// TIA Portal V20 program export: 4 tag tables, 69 data types, 13 data blocks, 100 code blocks (in call order from the OBs), 16 instance data blocks

VAR_GLOBAL   // PLC tag table "Default tag table"
END_VAR

VAR_GLOBAL   // PLC tag table "LKinCtrl_Configuration"
END_VAR
VAR_GLOBAL CONSTANT   // user constants
   LKINCTRL_SPTP_EXECUTION_STATUS_OUTPUT : Int := 0;   // 0: Regular time status; 1: Inverted time status; 2: Approximate cartesian distance
   LKINCTRL_LENGTH_OF_OFFSET_NAME : Int := 20;   // Length of offset name
   LKINCTRL_DISABLE_FLAG_RESET : Bool := TRUE;   // FALSE: Reset with execute & after done ; TRUE: No reset
   LKINCTRL_NO_OF_OFFSETS : Int := 3;   // Number of configurable offsets
   LKINCTRL_NO_OF_START_EXECUTE_CMDS : Int := 1;   // Number of cmds to be buffered in first cycle
   LKINCTRL_LENGTH_OF_CMDPOINT_NAME : Int := 30;   // Length of point name
   LKINCTRL_NO_OF_CONVEYOR : Int := 5;   // Number of configurable offsets
   LKINCTRL_NO_OF_SEQ_EXECUTE_CMDS : Int := 1;   // Number of cmds to be buffered after first cycle
   LKINCTRL_NO_OF_CMD_VALUEFLAGS : Int := 4;   // Number of LREAL flags per command
   LKINCTRL_NO_OF_ZONES : Int := 10;   // Number of zone definitions
   LKINCTRL_NO_OF_PATHDATA_ELEMENTS : Int := 200;   // Length of LKinCtrl_typePathData
   LKINCTRL_NO_OF_CMD_SETFLAGS : Int := 3;   // Number of Boolean flags per command
   LKINCTRL_LENGTH_OF_PATHDATA_NAME : Int := 20;   // Length of PathData name
   LKINCTRL_NO_OF_POINTS_AT_POINT_TABLE : Int := 30;   // Number of points at point table. Valid values are 1..x
   LKINCTRL_LENGTH_OF_TO_NAME : UInt := 30;   // Maximum number of characters for technology object name.
   LKINCTRL_NO_OF_LAST_VALUEFLAG : Int := 30;   // Number of value flags at MovePath FB
   LKINCTRL_NO_OF_LAST_SETFLAG : Int := 30;   // Number of flags at MovePath FB
   LKINCTRL_NO_OF_PATHS : Int := 5;   // Number of paths. Valid values are 1..x
END_VAR

VAR_GLOBAL   // PLC tag table "LKinCtrl_Constants"
END_VAR
VAR_GLOBAL CONSTANT   // user constants
   LKINCTRL_MC_MOVELINEARREL : Int := 2;   // cmdType for linear relative command
   LKINCTRL_FM_SET_BEFORE_AND_NO_RESET : USInt := 1;   // set flag before cmd and no reset
   LKINCTRL_MC_ACTIVATE_KIN_ZONE : Int := 34;   // cmdType for activating a workspace zone
   LKINCTRL_MC_MOVELINEARABS : Int := 1;   // cmdType for linear absolute command
   LKINCTRL_FM_SET_AFTER_AND_NO_RESET_AND_WAIT_FOR_ACKNOWLEDGE : USInt := 15;   // set flag after cmd and wait for external reset
   LKINCTRL_NO_OF_PATHDATA_PREBUFFER_ELEMENTS : Int := 5;   // number of PreBuffer elements
   LKINCTRL_FM_RESET_BEFORE : USInt := 20;   // reset flag at start of command
   LKINCTRL_FM_NO_SET_AND_WAIT_FOR_FALSE_ONCE : USInt := 25;   // do not set or reset flag but wait for flag to be false once during command
   LKINCTRL_TABLE_MASK_ARRAY_ENTRIES : DInt := 10;   // maximum size of searchable table
   LKINCTRL_CS_USER_FRAME_4 : Int := 14;   // select fourth user frame
   LKINCTRL_MC_MOVEDIRECTREL : Int := 6;   // cmdType for move direct relative command
   LKINCTRL_FM_DEACTIVATED : USInt := 0;   // flag deactiavted
   LKINCTRL_FM_SET_BEFORE_AND_RESET_AFTER_ONE_CYCLE : USInt := 3;   // set flag before cmd and reset after one cycle
   LKINCTRL_MC_SET_USER_FRAME : Int := 21;   // cmdType for set user frame
   LKINCTRL_CS_NO_OF_FIRST_USER_FRAME : Int := 11;   // index of first user frame
   LKINCTRL_CONFIG_END_OFFSET_COMP : Int := 40;   // cmdType for ending offset compensation
   LKINCTRL_CMD_WAIT_TIME : Int := 100;   // cmdType for wait time command
   LKINCTRL_COMP_RIGHT : Int := 2;   // tool radius compensation to the right
   LKINCTRL_MC_DEFINE_KIN_ZONE : Int := 33;   // cmdType for definining workspace zone
   LKINCTRL_MC_DESYNC_CONVEYOR : Int := 50;   // cmdType for conveyor desync
   LKINCTRL_MC_ACTIVATE_TOOL : Int := 23;   // cmdType for activating a tool
   LKINCTRL_MC_MOVECIRCULARABS : Int := 3;   // cmdType for circular absolute command
   LKINCTRL_CS_USER_FRAME_3 : Int := 13;   // select third user frame
   LKINCTRL_NO_OF_SETFLAGS_BUFFER_ELEMENTS : Int := 15;   // set as double of LKINCTRL_NO_OF_PATHDATA_PREBUFFER_ELEMENTS
   LKINCTRL_TABLE_TYPE_NONSELECTABLE : USInt := 2;   // constant for type non selectable table
   LKINCTRL_CS_USER_FRAME_2 : Int := 12;   // select second user frame
   LKINCTRL_CIRCMODE_GCODE : Int := 3;   // circMode used in GCode
   LKINCTRL_FM_SET_BEFORE_AND_NO_RESET_AND_WAIT_FOR_ACKNOWLEDGE : USInt := 5;   // set flag before cmd and wait for external reset
   LKINCTRL_CS_NO_OF_LAST_USER_FRAME : Int := 15;   // index of last user frame
   LKINCTRL_MC_ACTIVATE_WS_ZONE : Int := 31;   // cmdType for activating a workspace zone
   LKINCTRL_CS_USER_FRAME_1 : Int := 11;   // select first user frame
   LKINCTRL_MC_DEACTIVATE_WS_ZONE : Int := 32;   // cmdType for deactivating workspace zone
   LKINCTRL_FM_DISTANCE_TOLERANCE : LReal := 0.01;   // tolerance for flagmode 10
   LKINCTRL_CONFIG_START_OFFSET_COMP_LEFT : Int := 41;   // cmdType for starting offset compensation left
   LKINCTRL_FM_SET_BEFORE_AND_RESET_AFTER : USInt := 2;   // set flag before cmd and reset after
   LKINCTRL_MC_MOVECIRCULARREL : Int := 4;   // cmdType for circular relative command
   LKINCTRL_OUTER_CORNER : Int := 1;   // Outer corner (linear / linear intersection)
   LKINCTRL_INNER_CORNER : Int := 2;   // Inner corner (linear / linear intersection)
   LKINCTRL_FM_NO_SET_AND_WAIT_FOR_TRUE_ONCE : USInt := 26;   // do not set or reset flag but wait for flag to be true once during command
   LKINCTRL_MC_SHIFT_CS_REL : Int := 60;   // cmdType for relative shift of CS
   LKINCTRL_FM_SET_AT_REMAINING_DISTANCE : USInt := 10;   // set flag at remaining distance
   LKINCTRL_MC_DEACTIVATE_KIN_ZONE : Int := 35;   // cmdType for deactivating workspace zone
   LKINCTRL_COMP_LEFT : Int := 1;   // tool radius compensation to the left
   LKINCTRL_FM_SET_AFTER_AND_RESET_AFTER_ONE_CYCLE : USInt := 13;   // set flag after cmd and reset after one cycle
   LKINCTRL_CONFIG_START_OFFSET_COMP_RIGHT : Int := 42;   // cmdType for starting offset compensation right
   LKINCTRL_CS_USER_FRAME_5 : Int := 15;   // select fifth user frame
   LKINCTRL_TABLE_TYPE_SELECTABLE : USInt := 1;   // constant for type regular table
   LKINCTRL_MC_TRACKCONVEYORBELT : Int := 10;   // cmdType for track conveyor belt command
   LKINCTRL_NO_OF_VALID_BITS : Int := 6;   // number of valid bits in PathDataElement_advanced
   LKINCTRL_MC_SET_OCS_FRAME : Int := 20;   // cmdType for set frame command
   LKINCTRL_FM_SET_AFTER_AND_NO_RESET : USInt := 11;   // set flag after cmd and no reset
   LKINCTRL_MC_MOVEDIRECTABS : Int := 5;   // cmdType for move direct absolute command
   LKINCTRL_CMD_FLAG_ONLY : Int := 0;   // cmdType for flagOnly command (no motion)
   LKINCTRL_MC_DEFINE_WS_ZONE : Int := 30;   // cmdType for definining workspace zone
   LKINCTRL_MC_RESET_SHIFT : Int := 61;   // cmdType for resetting relative shift of CS
   LKINCTRL_FM_RESET_AFTER : USInt := 21;   // reset flag at end of command
   LKINCTRL_PI : LReal := 3.1415926535897932846264;   // constant value for pi
   LKINCTRL_FM_RESET_AT_REMAINING_DISTANCE : USInt := 22;   // reset flag if remaining distance of current command is reached
   LKINCTRL_MC_MOVELINEARPICKANDPLACE : Int := 11;   // cmdType for linear pick and place command sequence
   LKINCTRL_MC_SET_TOOL_FRAME : Int := 22;   // cmdType for defining tool frame
   LKINCTRL_DEFAULT_TO_NAME : WString := '- - -';   // Default name for technology objects
   LKINCTRL_KINEMATICS_TCS : DInt := 3;
   LKINCTRL_KINEMATICS_KINEMATICSZONES : DInt := 10;
   LKINCTRL_KINEMATICS_ZONE_STATE_VIOLATED : UInt := 3;   // Zone is valid, active and violated
   LKINCTRL_KINEMATICS_ZONE_STATE_INVALID : UInt := 0;   // Zone is invalid, inactive and not violated
   LKINCTRL_KINEMATICS_ZONE_STATE_VALID : UInt := 1;   // Zone is valid but not inactive and not violated
   LKINCTRL_KINEMATICS_WORKSPACEZONES : DInt := 10;
   LKINCTRL_KINEMATICS_OCS : DInt := 3;
   LKINCTRL_KINEMATICS_ZONE_STATE_ACTIVE : UInt := 2;   // Zone is valid and active but not violated
   LKINCTRL_KINEMATICS_CONVEYOR_TRACKING : UInt := 3;
   LKINCTRL_KINEMATICS_AXES : DInt := 6;
   LKINCTRL_MEAS_CMD_WITH_ACK : USInt := 2;   // continue after measurement command only with acknowledge
   LKINCTRL_MEAS_CMD_WO_ACK : USInt := 1;   // continue after measurement command without acknowledge
   LKINCTRL_DEFAULT_NAME : WString := '- - -';   // default name of points in datatype
   LKINCTRL_DEFAULT_NAME_STRING : String := '- - -';   // default name of strings in datatype
   LKINCTRL_NO_OF_PATHDATA_ELEMENTS_ADVANCED : Int := 200;   // LEGACY / Length of LKinCtrl_typePathData_advanced
   LKINCTRL_NO_OF_PATHDATA_ELEMENTS_REDUCED : Int := 10;   // LEGACY / Length of LKinCtrl_typePathData_reduced
END_VAR

VAR_GLOBAL   // PLC tag table "MC_Constants"
END_VAR
VAR_GLOBAL CONSTANT   // user constants
   DIRA_POSITIVE : Int := 1;   // Orientation direction 1: Positive direction
   DA_DEACTIVATED : Int := 0;   // Dynamic adaption 0: Deactivated
   CS_MCS : Int := 100;   // Coordinate system 100: Machine coordinate system (axis values)
   SM_ACTIVE_DYNAMICS : Int := 0;   // Stop mode 0: Stop with active dynamics
   LC_DEFAULT : DWord := 16#FFFFFFFF;   // LinkConstellation: Default to keep link constellation of kinematics
   CM_CENTER : Int := 1;   // Circle mode 1: "Arc" + "AuxPoint" defines circle center
   ZONE_DEACTIVATION_MODE_SIGNAL : DInt := 3;   // Zone deactivation mode 3: All signal zones
   BM_BLENDING_HIGH : Int := 5;   // Buffer mode 5: Blending with higher velocity
   BM_BUFFERED : Int := 1;   // Buffer mode 1: Standstill between motions
   PC_LONG_RUN_POSITIVE : Int := 2;   // Path choice 2: Longer positive circle segment
   IM_MAX_DYNAMICS : Int := 1;   // Interrupt mode 1: Interrupt with maximum dynamics
   CS_FCS : DInt := 0;   // Coordinate system 0: Flange coordinate system (FCS); Only valid for kinematics zone commands
   CS_TCS : DInt := 1;   // Coordinate system 1: Tool coordinate system (TCS); Only valid for kinematics zone commands
   DA_WITH_VARIABLE_LIMITS : Int := 1;   // Dynamic adaption 1: With segmentation of path
   DIRA_SHORTEST : Int := 3;   // Orientation direction 3: Shortest direction
   CS_OCS3 : Int := 3;   // Coordinate system 3: Object coordinate system 3 (OCS[3])
   CS_OCS1 : Int := 1;   // Coordinate system 1: Object coordinate system 1 (OCS[1])
   CM_RADIUS : Int := 2;   // Circle mode 2: "Radius" + "EndPoint" parameters define the circle segment
   CM_BORDER : Int := 0;   // Circle mode 0: "EndPoint" + "AuxPoint" parameter defines a point on circular path
   SM_MAX_DYNAMICS : Int := 1;   // Stop mode 1: Stop with maximum dynamics
   CP_XZ : Int := 0;   // Circle plane 0: Circle in X-Z plane
   CP_YZ : Int := 1;   // Circle plane 1: Circle in Y-Z plane
   IM_ACTIVE_DYNAMICS : Int := 0;   // Interrupt mode 0: Interrupt with active dynamics
   ZONE_DEACTIVATION_MODE_SPECIFIC : DInt := 0;   // Zone deactivation mode 0: Specific zone index
   BM_BLENDING_LOW : Int := 2;   // Buffer mode 2: Blending with lower velocity
   ZONE_DEACTIVATION_MODE_BLOCKED : DInt := 2;   // Zone deactivation mode 2: All blocked zones
   PC_NEGATIVE : Int := 1;   // Path choice 1: Shorter negative circle segment
   CP_XY : Int := 2;   // Circle plane 2: Circle in X-Y plane
   PM_ABS_ABS : DInt := 1;   // PositionMode 1: Interpretation of cartesian orientation as absolute (only effective for absolute MoveDirect commands)
   DA_WITH_CONSTANT_LIMITS : Int := 2;   // Dynamic adaption 2: No segmentation of path
   CS_OCS2 : Int := 2;   // Coordinate system 2: Object coordinate system 2 (OCS[2])
   CS_JCS : Int := 101;   // Coordinate system 101: Joint coordinate system (joint values)
   ZONE_DEACTIVATION_MODE_WORKSPACE : DInt := 4;   // Zone deactivation mode 4: Currently active workspace zone
   PM_ABS_REL : DInt := 2;   // PositionMode 2: Interpretation of cartesian orientation as relative (only effective for absolute MoveDirect commands)
   DIRA_NEGATIVE : Int := 2;   // Orientation direction 2: Negative direction
   CS_WCS : Int := 0;   // Coordinate system 0: World coordinate system (WCS)
   ZONE_DEACTIVATION_MODE_ALL : DInt := 1;   // Zone deactivation mode 1: All zones
   PC_POSITIVE : Int := 0;   // Path choice 0: Shorter positive circle segment
   PC_LONG_RUN_NEGATIVE : Int := 3;   // Path choice 3: Longer negative circle segment
   DA_DEFAULT : Int := -1;   // Dynamic adaption -1: Use default
END_VAR

TYPE "UDT_PathCmd"
TITLE = Buffered-path command element (V4.0 palletizing)
// One command in the buffered-path command list (GDB_PalletizingPath.aCmd). Authored by FB_AutoCtrl_Palletizing REGION 1, executed by REGION 4.
   STRUCT
      i16_CmdType : Int;   // Command type: 0 = END_OF_PATH, 1 = MOVE, 2 = GRIPPER, 3 = WAIT_ARRIVAL
      x : LReal;   // MOVE: target Cartesian X [mm]
      y : LReal;   // MOVE: target Cartesian Y [mm]
      z : LReal;   // MOVE: target Cartesian Z [mm]
      "a" : LReal;   // MOVE: target wrist orientation A [deg]
      lr_Velocity : LReal;   // MOVE: path velocity [mm/s]
      i16_BufferMode : Int;   // MOVE: MC_MoveLinearAbsolute BufferMode for this command -- 1 = stop at this point (BM_BUFFERED), 5 = blend through it (BM_BLENDING_HIGH). Never 0 (MC_Aborting is invalid for a kinematic path -> 16#80B2).
      lr_DwellMs : LReal;   // GRIPPER: grip/release settle hold time [ms]
      bo_GripperGrip : Bool;   // GRIPPER: level value written to GDB_Control.bo_gripperGrip
      bo_GripperRelease : Bool;   // GRIPPER: if TRUE, pulse GDB_Control.bo_gripperRelease for the dwell then drop it
      bo_IsBoxEnd : Bool;   // MOVE: TRUE on the PLACE_RETRACT move that completes a box -- increments statBoxesPlaced and re-arms the spawn request
      i16_HmiStep : Int;   // Value published to GDB_PalletizingCmd.i16_PalletStep when this command becomes active -- preserves the HMI 1..48 step display
   END_STRUCT;
END_TYPE

TYPE "UDT_Recipe"
TITLE = Box-product recipe (Module D)
// SCARA Phase 2 Module D recipe (2026-05-23). One flat box-product recipe: product L/W/H + gap, pallet base L/W + layer count, palletizing move dynamics. LPallPatt-shaped (typeProductData / typePalletData / typePnPDynamics, pruned for 1511T -- no block-packing, no mirroring, no interlayers, no multigripper). Consumed by FB_PatternAutoGen, which auto-fits a one-block grid and writes the result into GDB_PalletizingCmd's Module-C config members. PSC binds to GDB_ActiveRecipe.recipe.* member-for-member; the recipe library lives HMI-side on the panel.
   STRUCT
      sName : String[32];   // Recipe name (HMI display / identity).
      bo_Valid : Bool := FALSE;   // PSC handshake: PSC sets FALSE before transferring a parameter set and TRUE only after all members are written. FB_PatternAutoGen consumes the recipe only when this is TRUE -- closes the mid-write race that bites v9's recipe adapter.
      product : Struct
         lr_Length : LReal;   // Box length [mm]. Drives pitchX (= lr_Length + lr_Gap) via FB_PatternAutoGen.
         lr_Width : LReal;   // Box width [mm]. Drives pitchY (= lr_Width + lr_Gap).
         lr_Height : LReal;   // Box height [mm] -- copied straight to GDB_PalletizingCmd.lr_BoxHeight, the layer Z spacing for the Module-C builder.
         lr_Gap : LReal;   // Clearance between boxes [mm]; added to box dims to derive pitch. Set 0 for boxes edge-to-edge.
      END_STRUCT;
      pallet : Struct
         lr_BaseLength : LReal;   // Pallet base length [mm]. FB_PatternAutoGen auto-fits how many boxes fit along X: cols = (BaseLength + Gap) DIV (Length + Gap), floored.
         lr_BaseWidth : LReal;   // Pallet base width [mm]. FB_PatternAutoGen auto-fits how many boxes fit along Y: rows = (BaseWidth + Gap) DIV (Width + Gap), floored.
         i16_LayerCount : Int;   // Stacked layers (tower mode -- all layers use the same auto-gen grid). Total boxes = cols x rows x LayerCount, capped at the GDB_PalletizingPath.aCmd[] ceiling (22 for aCmd[1..200]).
      END_STRUCT;
      dynamics : Struct
         lr_Velocity : LReal;   // Palletizing-move path velocity [mm/s]. Written into GDB_PalletizingCmd.lr_MoveVelocity by FB_PatternAutoGen.
         lr_Acceleration : LReal;   // Palletizing-move acceleration [mm/s^2]. Written into GDB_PalletizingCmd.lr_MoveAccel.
         lr_Deceleration : LReal;   // Palletizing-move deceleration [mm/s^2]. Written into GDB_PalletizingCmd.lr_MoveDecel.
         lr_Jerk : LReal;   // Palletizing-move jerk [mm/s^3]. Written into GDB_PalletizingCmd.lr_MoveJerk.
      END_STRUCT;
   END_STRUCT;
END_TYPE

TYPE "UDT_typePoint5"
TITLE = SCARA TCP target point
// SCARA TCP target point (XYZA) for ABCDE 5-point cycle. Wang Shuo / Huashili pattern reference. B/C orientation omitted (SCARA 3D only supports A rotation about Z). / SCARA 末端目标点 (XYZA)，用于 ABCDE 5 点循环。王硕 / 华西丽模式参考。
   STRUCT
      x : LReal := 0.0;   // Cartesian X position [mm] / 笛卡尔 X 坐标 [mm]
      y : LReal := 0.0;   // Cartesian Y position [mm] / 笛卡尔 Y 坐标 [mm]
      z : LReal := 0.0;   // Cartesian Z position [mm] / 笛卡尔 Z 坐标 [mm]
      "a" : LReal := 0.0;   // Wrist orientation rotation A [deg] / 末端旋转角度 A [度]
   END_STRUCT;
END_TYPE

TYPE "UDT_typeMeasureInput"
   STRUCT
      input : Struct
         bo_Active : Bool;
         mode : Int;
      END_STRUCT;
      output : Struct
         done : Bool;
         busy : Bool;
         error : Bool;
         i32_ErrorCode : Word;
         r64_MeasuredValue1 : LReal;
         r64_MeasuredValue2 : LReal;
      END_STRUCT;
   END_STRUCT;
END_TYPE

TYPE "UDT_typePosCtrl"
   STRUCT
      input : Struct
         bo_estop : Bool;
         bo_enable : Bool;
         bo_reset : Bool;
         bo_home : Bool;
         bo_jogforward : Bool;
         bo_jogbackward : Bool;
         bo_movevelocity : Bool;
         bo_posabsolute : Bool;
         bo_posrelative : Bool;
         bo_gearin : Bool;
         bo_camin : Bool;
         bo_camout : Bool;
         bo_halt : Bool;
         bo_stop : Bool;
         configuration : Struct
            home { ExternalWritable := 'False'} : Struct
               i16_mode : Int;
               r64_homeposition : LReal;
               r64_ApproachVelocity : LReal := 10.0;
               r64_ReferencingVelocity : LReal := 5.0;
            END_STRUCT;
            jog : Struct
               r64_velocity : LReal := 5.0;
               r64_acceleration : LReal := 1000.0;
               r64_jerk : LReal := -1.0;
            END_STRUCT;
            movevelocity : Struct
               r64_velocity : LReal := 10.0;
               r64_acceleration : LReal := 1000.0;
               r64_jerk : LReal := -1.0;
               i16_direction : Int;
            END_STRUCT;
            posabsolute : Struct
               r64_velocity : LReal := 10.0;
               r64_position : LReal := 0.0;
               r64_acceleration : LReal := 1000.0;
               r64_jerk : LReal := -1.0;
               i16_direction : Int := 1;
            END_STRUCT;
            posrelative : Struct
               r64_velocity : LReal := 10.0;
               r64_position : LReal := 0.0;
               r64_acceleration : LReal := 1000.0;
               r64_jerk : LReal := -1.0;
            END_STRUCT;
            gearin : Struct
               RatioNumerator : DInt := 1;
               RatioDenominator : DInt := 1;
            END_STRUCT;
            camin : Struct
               i16_syncProfileReference : Int := 2;
               i16_applicationMode : Int := 0;
               r64_masterStartDistance : LReal;
               r64_masterSyncPosition : LReal;
               r64_masterOffset : LReal;
            END_STRUCT;
         END_STRUCT;
      END_STRUCT;
      output : Struct
         bo_communicationOk : Bool;
         bo_enabled : Bool;
         bo_homed : Bool;
         bo_inGear : Bool;
         bo_StarSync : Bool;
         bo_inSync : Bool;
         bo_fault : Bool;
         bo_endprofile : Bool;
         bo_SWLimitMinActived : Bool;
         bo_SWLimitMaxActived : Bool;
         bo_HWLimitMinActived : Bool;
         bo_HWLimitMaxActived : Bool;
         r64_actualVelocity : LReal;
         r64_actualPosition : LReal;
      END_STRUCT;
   END_STRUCT;
END_TYPE

TYPE "UDT_typeSpdCtrl"
   STRUCT
      input : Struct
         bo_enable : Bool := false;
         bo_estop : Bool := false;
         bo_reset : Bool := false;
         r32_speedSet : Real := 0.0;
         r32_torqueLimitSet : Real;
         r32_filterTime : Real := 100.0;
         tCycle : Real := 10.0;
         OBNum : Int := 30;
         HW_IO : HW_IO := 0;
         HW_IO_ADD : HW_IO;
         Reference : Struct
            r32_speed_Rpm : Real;
            r32_Torque_Nm : Real;
            r32_current_A : Real;
            r32_DCVolagte_V : Real;
            r32_power_Kw : Real;
            "r32_temperature_℃" : Real;
         END_STRUCT;
      END_STRUCT;
      output : Struct
         bo_enabled : Bool := false;
         bo_ready : Bool := false;
         bo_driveError : Bool := false;
         r32_actSpeed_Rpm : Real := 0.0;
         r32_actTorque_Nm : Real;
         r32_actCurrent_A : Real;
         r32_actDCVolagte_V : Real;
         r32_actPower_Kw : Real;
         "r32_actTemperature_℃" : Real;
         i16_warningCode : Word;
         i16_faultCode : Word;
      END_STRUCT;
   END_STRUCT;
END_TYPE

TYPE "UDT_typeKinCtrl"
   STRUCT
      input : Struct
         bo_estop : Bool;
         bo_enable : Bool;
         bo_reset : Bool;
         bo_home : Bool;
         jogframe : Struct
            "jogX+" : Bool;
            "jogX-" : Bool;
            "jogY+" : Bool;
            "jogY-" : Bool;
            "jogZ+" : Bool;
            "jogZ-" : Bool;
            "jogA+" : Bool;
            "jogA-" : Bool;
            "jogB+" : Bool;
            "jogB-" : Bool;
            "jogC+" : Bool;
            "jogC-" : Bool;
            bo_jogtoposition : Bool;
         END_STRUCT;
         bo_movepathstart : Bool;
         bo_movepathstop : Bool;
         bo_movepathhalt : Bool;
         configuration : Struct
            home { ExternalWritable := 'False'} : Struct
               i16_mode : Array[1..6] of Int;
               r64_homeposition : Array[1..6] of LReal;
            END_STRUCT;
            jogframe : Struct
               targetposition : Struct
                  x : LReal;
                  y : LReal;
                  z : LReal;
                  "a" : LReal;
                  "b" : LReal;
                  c : LReal;
               END_STRUCT;
               dynamics : "LKinCtrl_typeDynamics";   // Specification of the jog dynamics
            END_STRUCT;
         END_STRUCT;
      END_STRUCT;
      output : Struct
         bo_enabled : Bool;
         bo_homed : Bool;
         bo_fault : Bool;
         bo_done : Bool;
         i16_activeCmdNo : Int;
         actualposition : Struct
            x : LReal;
            y : LReal;
            z : LReal;
            "a" : LReal;
            "b" : LReal;
            c : LReal;
         END_STRUCT;
      END_STRUCT;
      inout : Struct
         PathData { S7_SetPoint := 'True'} : "LKinCtrl_typePathData";
      END_STRUCT;
   END_STRUCT;
   // input.configuration.jogframe.dynamics.sPTP.velocityFactor := -1.0;
   // input.configuration.jogframe.dynamics.sPTP.accelerationFactor := -1.0;
   // input.configuration.jogframe.dynamics.sPTP.decelerationFactor := -1.0;
   // input.configuration.jogframe.dynamics.sPTP.jerkFactor := -1.0;
END_TYPE

TYPE "LKinCtrl_bufferElement"
   STRUCT
      pathDataName : String["LKINCTRL_LENGTH_OF_PATHDATA_NAME"];
      pathDataIdentifier : USInt;
      setNumber : DInt;
      MotionType : Int := -1;
      MotionFBNo : Int;
      coordinateSystem : Int;
      transitionParameter : LReal;
      bufferMode : Int;
      measurementCmd : USInt;
      position : Array[1..6] of LReal;
   END_STRUCT;
END_TYPE

TYPE "LKinCtrl_typeAdvPointers"
   STRUCT
      addPointer : DInt := 0;   // pointer to add new comds to PathData after cmd has been executed by MovePath
      retrievePointer : DInt := 0;   // pointer to show which cmd is the next to be retrieved by MovePath
      addPointerRestarted : Bool;   // addPointer restarted after overflow
      ignoreAddPointer : Bool := TRUE;   // addPointer not taken into account for buffering, unless set by previous data source
      bufferLocked : Bool;   // buffer locked to wait for previous data source - read data locked
      preprocessingStop : Bool;   // parser reached a preprocessing stop
   END_STRUCT;
END_TYPE

TYPE "LKinCtrl_typeAuxFCDiagnostics"
TITLE = typeDiagnosticsFBTemplate
   STRUCT
      status : Word;   // Status of the FB or error identification when error occurred
      subfunctionStatus : Word;   // Status or return value of called FBs, FCs and system blocks
      axisNumber : Int;   // number of the corresponding axis the error occured in or a function effecting it
      errorDetail : UDInt;   // error detail of corresponding technology object the error occured in
      stateNumber : DInt;   // State in the state machine of the FB when the error occurred
   END_STRUCT;
END_TYPE

TYPE "LKinCtrl_typeCartesianPosition"
   STRUCT
      x : LReal;   // X
      y : LReal;   // Y
      z : LReal;   // Z
      "a" : LReal;   // A
      "b" : LReal;   // B
      c : LReal;   // C
   END_STRUCT;
END_TYPE

TYPE "LKinCtrl_typeCircleParameters"
   STRUCT
      circMode : DInt := 0;   // 0: auxPoint defines point on circle line; 1: auxPoint defines circle center; 2: radius and endPoint define circle segment; 3: GCode notation (end & aux point)
      point : DInt := -1;   // reference to point table, used for auxPoint
      auxPoint : Array[1..3] of LReal;   // auxiliary point for circle definition
      pathChoice : DInt := 0;   // circMode(0): not relevant; circMode(1): 0: pos direction; 1: neg direction; circMode(2): 0: short pos segment; 1: short neg segment; 2: long pos segment; 3: long neg segment
      circlePlane : DInt;   // circMode(0): not relevant; circMode(1+2): 0: XZ; 1: YZ; 2: XY
      radius : LReal;   // only in combination with circMode(2): radius
      arc : LReal;   // only in combination with circMode(1): arc
   END_STRUCT;
END_TYPE

TYPE "LKinCtrl_typeCmdLoggerElement"
   STRUCT
      cmdType : Int := -1;   // 1: MoveLinAbs; 2: MoveLinRel; 3: MoveCircAbs; 4: MoveCircRel; 5: MoveDirectAbs; 6: MoveDirectRel; 10: TrackConveyorBelt; 100: WaitTime; 40/41/42: ContourOffset; 0: FlagOnlyCmd; -1: End of List
      pathDataName : String["LKINCTRL_LENGTH_OF_PATHDATA_NAME"];   // name of PathData
      pathDataIdentifier : Int;   // identifier of PathData containing command
      cmdID : DInt;   // to be set to PathDataOperate[list position] by PreBuffer for identification in ExecuteBuffer
      cmdName : String[4];   // command name
      coordinateX : LReal;   // X (linear) / endPoint[1] (circular)
      coordinateY : LReal;   // Y (linear) / endPoint[2] (circular)
      coordinateZ : LReal;   // Z (linear) / endPoint[3] (circular)
      coordinateA : LReal;   // A (linear) / endPoint[4] (circular)
      coordSystem : DInt := 0;   // 0: WCS; 1: OCS[1]; 2: OCS[2]; 3: OCS[3]
      bufferMode : DInt := 1;   // 1: standstill between commands, 2: blending with lower speed; 5: blending with higher speed
      transitionParameter : LReal;   // blending distance - >0.0: configured value used; <0.0: maximum possible blending distance used
      dynVelocity : LReal;   // >0.0: configured value used; <0.0: default TO setting used
      dynAcceleration : LReal;   // >0.0: configured value used; <0.0: default TO setting used
      dynDeceleration : LReal;   // >0.0: configured value used; <0.0: default TO setting used
      dynJerk : LReal;   // >0.0: configured value used; <0.0: default TO setting used
      dynamicAdpation : DInt;   // <0.0: default TO setting used; 0: no dynamic adaption; 1: with variable limits; 2: with constant limits
      linkConstellation : DWord;   // linkConstellation (effective for MoveDirect commands only)
      positionMode : DInt;   // 1: absolute cartesian position and absolute orientation; 2: absolute cartesian position and relative orientation (effective for MoveDirect commands only)
      circMode : DInt;   // 0: auxPoint defines point on circle line; 1: auxPoint defines circle center; 2: radius and endPoint define circle segment
      auxPoint_1 : LReal;   // auxiliary point for circle definition
      auxPoint_2 : LReal;   // auxiliary point for circle definition
      auxPoint_3 : LReal;   // auxiliary point for circle definition
      pathChoice : DInt;   // circMode(0): not relevant; circMode(1): 0: pos direction; 1: neg direction; circMode(2): 0: short pos segment; 1: short neg segment; 2: long pos segment; 3: long neg segment
      circlePlane : DInt;   // circMode(0): not relevant; circMode(1+2): 0: XZ; 1: YZ; 2: XY
      radius : LReal;   // only in combination with circMode(2): radius
      arc : LReal;   // only in combination with circMode(1): arc
   END_STRUCT;
END_TYPE

TYPE "LKinCtrl_typeConfiguration"
   STRUCT
      offsetParameter : Array[1.."LKINCTRL_NO_OF_OFFSETS"] of "LKinCtrl_typeContourOffsetParameter";   // offset parameter settings
      conveyorParameter : Array[1.."LKINCTRL_NO_OF_CONVEYOR"] of "LKinCtrl_typeConveyorConfiguration";   // conveyor parameter settings
      userFrames : Array["LKINCTRL_CS_NO_OF_FIRST_USER_FRAME".."LKINCTRL_CS_NO_OF_LAST_USER_FRAME"] of "LKinCtrl_typeFrame";   // user frames configuration
      workspaceZones : Array[1.."LKINCTRL_NO_OF_ZONES"] of "LKinCtrl_typeWorkspaceZoneDefinition";   // workspace zone configurations
      kinematicsZones : Array[1.."LKINCTRL_NO_OF_ZONES"] of "LKinCtrl_typeKinematicsZoneDefinition";   // kinematics zone configuration
      stopMode : DInt;   // MC_GroupStop dynamics; 0: stop with dynamics of active motion job; 1: stop with maximum kinematics dynamics (dynamics adaption still effective); 10: stop with dynamics of active motion job and desync conveyor; 11: stop with maximum kinematics dynamics and desync conveyor
      interruptMode : DInt;   // MC_GroupInterrupt dynamics; 0: interrupt with dynamics of active motion job; 1: interrupt with maximum kinematics dynamics (dynamics adaption still effective)
   END_STRUCT;
END_TYPE

TYPE "LKinCtrl_typeConfigurationAxis"
   STRUCT
      "name" { ExternalAccessible := 'False'; ExternalVisible := 'False'; ExternalWritable := 'False'; S7_SetPoint := 'True'} : WString["LKINCTRL_LENGTH_OF_TO_NAME"];   // Axis name shown on HMI
      used { ExternalAccessible := 'False'; ExternalVisible := 'False'; ExternalWritable := 'False'; S7_SetPoint := 'True'} : Bool := FALSE;   // TRUE: Axis is used (only relevant for additional axes, kinematic axes are always used)
      withBrake { ExternalAccessible := 'False'; ExternalVisible := 'False'; ExternalWritable := 'False'; S7_SetPoint := 'True'} : Bool := FALSE;   // TRUE: Axis has a motor holding brake
      homePosition { ExternalAccessible := 'False'; ExternalVisible := 'False'; ExternalWritable := 'False'; S7_SetPoint := 'True'} : LReal := 0.0;   // Defines the default homing position
      coupling { ExternalAccessible := 'False'; ExternalVisible := 'False'; ExternalWritable := 'False'; S7_SetPoint := 'True'} : Bool := FALSE;   // TRUE: Coupling present
      jog { ExternalAccessible := 'False'; ExternalVisible := 'False'; ExternalWritable := 'False'; S7_SetPoint := 'True'} : "LKinCtrl_typeJogConfiguration";
   END_STRUCT;
   // jog.accelerationTime := 0.2;
   // jog.maxVelocityManual := 10.0;
   // jog.maxVelocityTestRun := 10.0;
   // jog.presetIncrementCoarse := 5.0;
   // jog.presetIncrementFine := 1.0;
   // jog.presetIncrementPrecise := 0.5;
END_TYPE

TYPE "LKinCtrl_typeConfigurationKinematics"
   STRUCT
      "name" { ExternalAccessible := 'False'; ExternalVisible := 'False'; ExternalWritable := 'False'; S7_SetPoint := 'True'} : WString["LKINCTRL_LENGTH_OF_TO_NAME"];
      jogPath { ExternalAccessible := 'False'; ExternalVisible := 'False'; ExternalWritable := 'False'; S7_SetPoint := 'True'} : "LKinCtrl_typeJogConfiguration";
      jogOrientation { ExternalAccessible := 'False'; ExternalVisible := 'False'; ExternalWritable := 'False'; S7_SetPoint := 'True'} : "LKinCtrl_typeJogConfiguration";
   END_STRUCT;
   // jogPath.accelerationTime := 0.2;
   // jogPath.maxVelocityManual := 250.0;
   // jogPath.maxVelocityTestRun := 250.0;
   // jogPath.presetIncrementCoarse := 10.0;
   // jogPath.presetIncrementFine := 1.0;
   // jogPath.presetIncrementPrecise := 0.1;
   // jogOrientation.accelerationTime := 0.2;
   // jogOrientation.maxVelocityManual := 10.0;
   // jogOrientation.maxVelocityTestRun := 10.0;
   // jogOrientation.presetIncrementCoarse := 5.0;
   // jogOrientation.presetIncrementFine := 1.0;
   // jogOrientation.presetIncrementPrecise := 0.1;
END_TYPE

TYPE "LKinCtrl_typeContourOffsetParameter"
   STRUCT
      "name" : String["LKINCTRL_LENGTH_OF_OFFSET_NAME"];   // offset name
      radius : LReal;   // offset radius
      length : LReal;   // offset length
   END_STRUCT;
END_TYPE

TYPE "LKinCtrl_typeConveyorConfiguration"
   STRUCT
      conveyorBeltAxis : DB_ANY;   // Conveyor belt axis DB
      conveyorBeltOrigin : TO_Struct_Kinematics_Frame;   // Frame to origin of conveyor belt
      initialObjectPosition : TO_Struct_Kinematics_Frame;   // Initial object position on conveyor (only x allowed)
   END_STRUCT;
END_TYPE

TYPE "LKinCtrl_typeConveyorParameter"
   STRUCT
      conveyorParaNo : DInt := 0;   // selection of conveyor parameter set from configuration structure
   END_STRUCT;
END_TYPE

TYPE "LKinCtrl_typeDiagnosticsPathSelect"
TITLE = typeDiagnosticsFBTemplate
   STRUCT
      status : Word;   // Status of the FC or error identification when error occurred
      entryID : Int;   // identifier for false entry
   END_STRUCT;
END_TYPE

TYPE "LKinCtrl_typeDynamics"
   STRUCT
      path : "LKinCtrl_typePathDynamics";   // Specification of the path dynamics
      orientation : "LKinCtrl_typePathDynamics";   // Specification of the orientation dynamics
      dynamicAdaption : DInt := 1;   // 0=no dynamic adaption, 1=dynamic adaptation with segmentation of the path, 2=dynamic adaptation without segmentation of the path
      directionA : DInt := 3;   // 1=positive direction, 2=negative direction, 3=shortest distance
      sPTP : "LKinCtrl_typeSPTPDynamics";   // Specification of the dynamic factor for sptp movement
   END_STRUCT;
END_TYPE

TYPE "LKinCtrl_typeExecuteKinMotionCmdDiagnostics"
   STRUCT
      status : Word;   // status of the FB
      faultPathDataName : String["LKINCTRL_LENGTH_OF_PATHDATA_NAME"];   // number of PathData with occurring error in PathData set
      faultSetNumber : DInt;   // number of PathData set with occurring error
      faultFBNumber : DInt;   // number of motionCommand FB with occurring error
      motionFBstatus : DWord;   // status of motion FB (internal) an error occurred in
      stateMachine : Int;   // stateMachine status
      kinematicsStatusWord : DWord;   // statusWord TO kinematics
      kinematicsErrorWord : DWord;   // errorWord TO kinematics
   END_STRUCT;
END_TYPE

TYPE "LKinCtrl_typeFlagBufferElement"
   STRUCT
      pathDataName : String["LKINCTRL_LENGTH_OF_PATHDATA_NAME"] := '';   // PathData name of specific command
      pathDataIdentifier : DInt;   // PathData identifier counter of specific command
      cmdId : DInt := 0;   // cmdId of command in PathData
      isIntermediateCmd : Bool;   // TRUE: command is intermediate command
      setFlags : Array[1.."LKINCTRL_NO_OF_CMD_SETFLAGS"] of "LKinCtrl_typeSetFlagElement_Bool";   // setFlags structure equal to PathData command entry
      valueFlags : Array[1.."LKINCTRL_NO_OF_CMD_VALUEFLAGS"] of "LKinCtrl_typeSetFlagElement_LReal";   // setFlags structure equal to PathData command entry
   END_STRUCT;
END_TYPE

TYPE "LKinCtrl_typeFrame"
   STRUCT
      x : LReal;   // Translation in x
      y : LReal;   // Translation in y
      z : LReal;   // Translation in z
      "a" : LReal;   // Rotation around z axis
      "b" : LReal;   // Rotation around y axis
      c : LReal;   // Roataion around x axis
   END_STRUCT;
END_TYPE

TYPE "LKinCtrl_typeJogConfiguration"
   STRUCT
      accelerationTime { ExternalAccessible := 'False'; ExternalVisible := 'False'; ExternalWritable := 'False'; S7_SetPoint := 'True'} : LReal;
      maxVelocityManual { ExternalAccessible := 'False'; ExternalVisible := 'False'; ExternalWritable := 'False'; S7_SetPoint := 'True'} : LReal;
      maxVelocityTestRun { ExternalAccessible := 'False'; ExternalVisible := 'False'; ExternalWritable := 'False'; S7_SetPoint := 'True'} : LReal;
      presetIncrementCoarse { ExternalAccessible := 'False'; ExternalVisible := 'False'; ExternalWritable := 'False'; S7_SetPoint := 'True'} : LReal;
      presetIncrementFine { ExternalAccessible := 'False'; ExternalVisible := 'False'; ExternalWritable := 'False'; S7_SetPoint := 'True'} : LReal;
      presetIncrementPrecise { ExternalAccessible := 'False'; ExternalVisible := 'False'; ExternalWritable := 'False'; S7_SetPoint := 'True'} : LReal;
   END_STRUCT;
END_TYPE

TYPE "LKinCtrl_typeJogFrameDiagnostics"
// support: tech.team.motioncontrol@siemens.com
   STRUCT
      timeStamp : Date_And_Time;   // Time stamp at which the error occurred
      status : Word;   // Status of FB when error occurred
      stateNumber : DInt;   // State in the state machine of the FB when the error occurred
   END_STRUCT;
END_TYPE

TYPE "LKinCtrl_typeKinematicsZoneDefinition"
   STRUCT
      coordinateSystem : DInt;   // 0:FCS, 1:TCS
      frame : "LKinCtrl_typeFrame";   // shifting of the zone zero point in relation to the reference system
      geometryType : DInt;   // 0:Cuboid, 1:Sphere, 2:Cylinder
      geometryParameter : Array[1..3] of LReal;   // geometry parameter depending on geometry type
   END_STRUCT;
END_TYPE

TYPE "LKinCtrl_typeMoveDirectParameter"
   STRUCT
      linkConstellation : DWord := 16#FFFF_FFFF;   // linkConstellation (effective for MoveDirect commands only)
      positionMode : DInt := 1;   // 1: absolute cartesian position and absolute orientation; 2: absolute cartesian position and relative orientation (effective for MoveDirect commands only)
      turnJoint : Array[1..6] of DInt;   // turn joint setting (effective for MoveDirect commands only)
   END_STRUCT;
END_TYPE

TYPE "LKinCtrl_typeMovePathDiagnostics"
   STRUCT
      errorID : Word;   // errorID of the FB
      pathDataName : String["LKINCTRL_LENGTH_OF_PATHDATA_NAME"];   // name of PathData an error occurred in
      cmdNumber : DInt;   // command number (in PathData) an error occurred in
      stateMovePath : DInt;   // state machine status FB
      statusSubFunction : Word;   // status of LKinCtrl_MC_ExecuteKinMotionCmd
      motionFBNumber : DInt;   // motion FB number (internal) an error occurred in
      motionFBStatus : DWord;   // status of motion FB (internal) an error occurred in
      kinematicsStatusWord : DWord;   // statusWord TO kinematics
      kinematicsErrorWord : DWord;   // errorWord TO kinematics
   END_STRUCT;
END_TYPE

TYPE "LKinCtrl_typeMovePickAndPlaceParameters"
   STRUCT
      startParameter : "LKinCtrl_typePnPParameter";   // Start vector parameter
      targetParameter : "LKinCtrl_typePnPParameter";   // Target vector parameter
   END_STRUCT;
END_TYPE

TYPE "LKinCtrl_typePathData"
   STRUCT
      pathDataName : String["LKINCTRL_LENGTH_OF_PATHDATA_NAME"];   // name of PathData
      LKinLangInterface : "LKinCtrl_typeAdvPointers";   // pointers to add / retrieve cmds in PathData
      commands : Array[1.."LKINCTRL_NO_OF_PATHDATA_ELEMENTS"] of "LKinCtrl_typePathDataElement";   // command list
   END_STRUCT;
   // commands[1].cmdParameters.transitionParameters[1] := -1.0;
   // commands[2].cmdParameters.transitionParameters[1] := -1.0;
   // commands[3].cmdParameters.transitionParameters[1] := -1.0;
   // commands[4].cmdParameters.transitionParameters[1] := -1.0;
   // commands[5].cmdParameters.transitionParameters[1] := -1.0;
   // commands[6].cmdParameters.transitionParameters[1] := -1.0;
   // commands[7].cmdParameters.transitionParameters[1] := -1.0;
   // commands[8].cmdParameters.transitionParameters[1] := -1.0;
   // commands[9].cmdParameters.transitionParameters[1] := -1.0;
   // commands[10].cmdParameters.transitionParameters[1] := -1.0;
   // commands[11].cmdParameters.transitionParameters[1] := -1.0;
   // commands[12].cmdParameters.transitionParameters[1] := -1.0;
   // commands[13].cmdParameters.transitionParameters[1] := -1.0;
   // commands[14].cmdParameters.transitionParameters[1] := -1.0;
   // commands[15].cmdParameters.transitionParameters[1] := -1.0;
   // commands[16].cmdParameters.transitionParameters[1] := -1.0;
   // commands[17].cmdParameters.transitionParameters[1] := -1.0;
   // commands[18].cmdParameters.transitionParameters[1] := -1.0;
   // commands[19].cmdParameters.transitionParameters[1] := -1.0;
   // commands[20].cmdParameters.transitionParameters[1] := -1.0;
END_TYPE

TYPE "LKinCtrl_typePathDataElement"
   STRUCT
      cmdType : Int := -1;   // 1: MoveLinAbs; 2: MoveLinRel; 3: MoveCircAbs; 4: MoveCircRel; 5: MoveDirectAbs; 6: MoveDirectRel; 10: TrackConveyorBelt; 100: WaitTime; 40/41/42: ContourOffset; 0: FlagOnlyCmd; -1: End of List; 20-23: Frame cmds; 30-35: Zone cmds
      cmdActivated : Bool := TRUE;   // (de)activation of command
      cmdName : String["LKINCTRL_LENGTH_OF_CMDPOINT_NAME"];   // name of command
      point : DInt := -1;   // reference to point table, used for cmdCoordinates
      measurementCmd : USInt;   // 0: deactivated; 1: without acknowledge; 2: with acknowledge
      cmdCoordinates : "LKinCtrl_typePointCoordinates";   // target coordinate definition
      cmdParameters : "LKinCtrl_typePointParameter";   // additional command parameters
      setFlags : Array[1.."LKINCTRL_NO_OF_CMD_SETFLAGS"] of "LKinCtrl_typeSetFlagElement_Bool";   // flags to control actuators
      valueFlags : Array[1.."LKINCTRL_NO_OF_CMD_VALUEFLAGS"] of "LKinCtrl_typeSetFlagElement_LReal";   // value flags to control actuators
      parameterValid : Array[1.."LKINCTRL_NO_OF_VALID_BITS"] of Bool;
   END_STRUCT;
   // cmdParameters.transitionParameters[1] := -1.0;
   // parameterValid[1..6] := TRUE;
END_TYPE

TYPE "LKinCtrl_typePathDataElement_PreBuf"
   STRUCT
      pathDataName : String["LKINCTRL_LENGTH_OF_PATHDATA_NAME"];   // name of PathData
      pathDataIdentifier : USInt;   // identifier of PathData
      isIntermediateCmd : Bool;   // TRUE: command is intermediate command
      cmdID : DInt;   // to be set to PathDataOperate[list position] by PreBuffer for identification in ExecuteBuffer
      cmdType : Int := -1;   // 1: MoveLinAbs; 2: MoveLinRel; 3: MoveCircAbs; 4: MoveCircRel; 5: MoveDirectAbs; 6: MoveDirectRel; 10: TrackConveyorBelt; 100: WaitTime; 40/41/42: ContourOffset; 0: FlagOnlyCmd; -1: End of List; 20-23: Frame cmds; 30-35: Zone cmds
      cmdName : String["LKINCTRL_LENGTH_OF_CMDPOINT_NAME"];   // command name
      measurementCmd : USInt;   // 0: deactivated; 1: without acknowledge; 2: with acknowledge
      cmdCoordinates : "LKinCtrl_typePointCoordinates_PreBuf";   // command coordinates
      cmdParameters : "LKinCtrl_typePointParameter";   // command parameters
      setFlags : Array[1.."LKINCTRL_NO_OF_CMD_SETFLAGS"] of "LKinCtrl_typeSetFlagElement_Bool";   // flags to control actuators
      valueFlags : Array[1.."LKINCTRL_NO_OF_CMD_VALUEFLAGS"] of "LKinCtrl_typeSetFlagElement_LReal";   // value flags to control actuators
      parameterValid : Array[1.."LKINCTRL_NO_OF_VALID_BITS"] of Bool;   // valid bit for cartesian position parameters
   END_STRUCT;
   // cmdParameters.transitionParameters[1] := -1.0;
   // parameterValid[1..6] := TRUE;
END_TYPE

TYPE "LKinCtrl_typePathDataElement_advanced"
   STRUCT
      cmdType : Int := -1;   // 1: MoveLinAbs; 2: MoveLinRel; 3: MoveCircAbs; 4: MoveCircRel; 5: MoveDirectAbs; 6: MoveDirectRel; 10: TrackConveyorBelt; 100: WaitTime; 40/41/42: ContourOffset; 0: FlagOnlyCmd; -1: End of List; 20-23: Frame cmds; 30-35: Zone cmds
      cmdActivated : Bool := TRUE;   // (de)activation of command
      cmdName : String["LKINCTRL_LENGTH_OF_CMDPOINT_NAME"];   // name of command
      point : DInt := -1;   // reference to point table, used for cmdCoordinates
      measurementCmd : USInt;   // 0: deactivated; 1: without acknowledge; 2: with acknowledge
      cmdCoordinates : "LKinCtrl_typePointCoordinates";   // target coordinate definition
      cmdParameters : "LKinCtrl_typePointParameter";   // additional command parameters
      setFlags : Array[1.."LKINCTRL_NO_OF_CMD_SETFLAGS"] of "LKinCtrl_typeSetFlagElement_Bool";   // flags to control actuators
      valueFlags : Array[1.."LKINCTRL_NO_OF_CMD_VALUEFLAGS"] of "LKinCtrl_typeSetFlagElement_LReal";   // value flags to control actuators
      parameterValid : Array[1.."LKINCTRL_NO_OF_VALID_BITS"] of Bool;   // valid bit for cartesian position parameters
   END_STRUCT;
   // cmdParameters.transitionParameters[1] := -1.0;
   // parameterValid[1..6] := TRUE;
END_TYPE

TYPE "LKinCtrl_typePathDataElement_reduced"
   STRUCT
      cmdType : Int := -1;   // 1: MoveLinAbs; 2: MoveLinRel; 100: WaitTime; 0: FlagOnlyCmd; -1: End of List
      cmdActivated : Bool := TRUE;   // (de)activation of command
      cmdName : String["LKINCTRL_LENGTH_OF_CMDPOINT_NAME"];   // name of command
      point : DInt := -1;   // reference to point table, used for cmdCoordinates
      cmdCoordinates : "LKinCtrl_typePointCoordinates";   // target coordinate definition
      cmdParameters : "LKinCtrl_typePointParameter_reduced";   // additional command parameters
      setFlags : Array[1.."LKINCTRL_NO_OF_CMD_SETFLAGS"] of "LKinCtrl_typeSetFlagElement_Bool";   // flags to control actuators
      valueFlags : Array[1.."LKINCTRL_NO_OF_CMD_VALUEFLAGS"] of "LKinCtrl_typeSetFlagElement_LReal";   // value flags to control actuators
   END_STRUCT;
   // cmdParameters.transitionParameters[1] := -1.0;
END_TYPE

TYPE "LKinCtrl_typePathData_PreBuf"
   STRUCT
      pathDataName : String["LKINCTRL_LENGTH_OF_PATHDATA_NAME"];   // name of PathData
      commands : Array[1.."LKINCTRL_NO_OF_PATHDATA_PREBUFFER_ELEMENTS"] of "LKinCtrl_typePathDataElement_PreBuf";   // command list
      addPointer : Int;   // pointer marking slot for adding of next command in PathDataPreBuffered
      retrievePointer : Int;   // pointer marking command entry to be read in PathDataPreBuffered
      addPointerRestarted : Bool;   // addPointer restarted after overflow
   END_STRUCT;
   // commands[1].cmdParameters.transitionParameters[1] := -1.0;
   // commands[2].cmdParameters.transitionParameters[1] := -1.0;
   // commands[3].cmdParameters.transitionParameters[1] := -1.0;
   // commands[4].cmdParameters.transitionParameters[1] := -1.0;
   // commands[5].cmdParameters.transitionParameters[1] := -1.0;
   // commands[1].parameterValid[1..4] := TRUE;
   // commands[2].parameterValid[1..4] := TRUE;
   // commands[3].parameterValid[1..4] := TRUE;
   // commands[4].parameterValid[1..4] := TRUE;
   // commands[5].parameterValid[1..4] := TRUE;
END_TYPE

TYPE "LKinCtrl_typePathData_advanced"
   STRUCT
      pathDataName : String["LKINCTRL_LENGTH_OF_PATHDATA_NAME"];   // name of PathData
      pointers : "LKinCtrl_typeAdvPointers";   // pointers to add / retrieve cmds in PathData
      commands : Array[1.."LKINCTRL_NO_OF_PATHDATA_ELEMENTS_ADVANCED"] of "LKinCtrl_typePathDataElement_advanced";   // command list
   END_STRUCT;
   // commands[1].cmdParameters.transitionParameters[1] := -1.0;
   // commands[2].cmdParameters.transitionParameters[1] := -1.0;
   // commands[3].cmdParameters.transitionParameters[1] := -1.0;
   // commands[4].cmdParameters.transitionParameters[1] := -1.0;
   // commands[5].cmdParameters.transitionParameters[1] := -1.0;
   // commands[6].cmdParameters.transitionParameters[1] := -1.0;
   // commands[7].cmdParameters.transitionParameters[1] := -1.0;
   // commands[8].cmdParameters.transitionParameters[1] := -1.0;
   // commands[9].cmdParameters.transitionParameters[1] := -1.0;
   // commands[10].cmdParameters.transitionParameters[1] := -1.0;
   // commands[11].cmdParameters.transitionParameters[1] := -1.0;
   // commands[12].cmdParameters.transitionParameters[1] := -1.0;
   // commands[13].cmdParameters.transitionParameters[1] := -1.0;
   // commands[14].cmdParameters.transitionParameters[1] := -1.0;
   // commands[15].cmdParameters.transitionParameters[1] := -1.0;
   // commands[16].cmdParameters.transitionParameters[1] := -1.0;
   // commands[17].cmdParameters.transitionParameters[1] := -1.0;
   // commands[18].cmdParameters.transitionParameters[1] := -1.0;
   // commands[19].cmdParameters.transitionParameters[1] := -1.0;
   // commands[20].cmdParameters.transitionParameters[1] := -1.0;
   // commands[1].parameterValid[1..4] := TRUE;
   // commands[2].parameterValid[1..4] := TRUE;
   // commands[3].parameterValid[1..4] := TRUE;
   // commands[4].parameterValid[1..4] := TRUE;
   // commands[5].parameterValid[1..4] := TRUE;
   // commands[6].parameterValid[1..4] := TRUE;
   // commands[7].parameterValid[1..4] := TRUE;
   // commands[8].parameterValid[1..4] := TRUE;
   // commands[9].parameterValid[1..4] := TRUE;
   // commands[10].parameterValid[1..4] := TRUE;
   // commands[11].parameterValid[1..4] := TRUE;
   // commands[12].parameterValid[1..4] := TRUE;
   // commands[13].parameterValid[1..4] := TRUE;
   // commands[14].parameterValid[1..4] := TRUE;
   // commands[15].parameterValid[1..4] := TRUE;
   // commands[16].parameterValid[1..4] := TRUE;
   // commands[17].parameterValid[1..4] := TRUE;
   // commands[18].parameterValid[1..4] := TRUE;
   // commands[19].parameterValid[1..4] := TRUE;
   // commands[20].parameterValid[1..4] := TRUE;
END_TYPE

TYPE "LKinCtrl_typePathData_reduced"
   STRUCT
      pathDataName : String["LKINCTRL_LENGTH_OF_PATHDATA_NAME"];   // name of PathData
      commands : Array[1.."LKINCTRL_NO_OF_PATHDATA_ELEMENTS_REDUCED"] of "LKinCtrl_typePathDataElement_reduced";   // command list
   END_STRUCT;
   // commands[1].cmdParameters.transitionParameters[1] := -1.0;
   // commands[2].cmdParameters.transitionParameters[1] := -1.0;
   // commands[3].cmdParameters.transitionParameters[1] := -1.0;
   // commands[4].cmdParameters.transitionParameters[1] := -1.0;
   // commands[5].cmdParameters.transitionParameters[1] := -1.0;
   // commands[6].cmdParameters.transitionParameters[1] := -1.0;
   // commands[7].cmdParameters.transitionParameters[1] := -1.0;
   // commands[8].cmdParameters.transitionParameters[1] := -1.0;
   // commands[9].cmdParameters.transitionParameters[1] := -1.0;
   // commands[10].cmdParameters.transitionParameters[1] := -1.0;
END_TYPE

TYPE "LKinCtrl_typePathDynamics"
   STRUCT
      velocity : LReal := -1.0;   // >0.0: configured value used; <0.0: default TO setting used; for cmdType = 100 ==> waitTime in ms
      acceleration : LReal := -1.0;   // >0.0: configured value used; <0.0: default TO setting used
      deceleration : LReal := -1.0;   // >0.0: configured value used; <0.0: default TO setting used
      jerk : LReal := -1.0;   // >0.0: configured value used; <0.0: default TO setting used
   END_STRUCT;
END_TYPE

TYPE "LKinCtrl_typePoint"
   STRUCT
      "name" : WString["LKINCTRL_LENGTH_OF_CMDPOINT_NAME"];   // Specification of a point name
      position : Array[0..5] of LReal;   // Specification of Cartesian position for a point
      coordSystem : USInt;   // Specification of a point coordinate system
      linkConstellation : DWord := 16#FFFF_FFFF;   // Specification of the target link constellation
      turnJoint : Array[0..5] of DInt;   // Only relevant with more than four interpolating kinematics axes - When "CoordSystem" = 0, 1, 2 or 3: target joint position range of the joint J[1..6]
   END_STRUCT;
END_TYPE

TYPE "LKinCtrl_typePointCoordinates"
   STRUCT
      cartesianPosition : "LKinCtrl_typeCartesianPosition";   // cartesian position
      coordSystem : DInt := 0;   // 0: WCS; 1: OCS[1]; 2: OCS[2]; 3: OCS[3]; 100: MCS
   END_STRUCT;
END_TYPE

TYPE "LKinCtrl_typePointCoordinates_PreBuf"
   STRUCT
      startPosition : Array[1..6] of LReal;   // absolute start position
      targetPosition : Array[1..6] of LReal;   // end position or relative distance depending on command type
      targetDistance : Array[1..6] of LReal;
      coordSystem : DInt := 0;   // 0: WCS; 1: OCS[1]; 2: OCS[2]; 3: OCS[3]
   END_STRUCT;
END_TYPE

TYPE "LKinCtrl_typePointParameter"
   STRUCT
      pathDynamics : "LKinCtrl_typePathDynamics";   // path dynamics for this command
      orientationDynamics : "LKinCtrl_typePathDynamics";   // orientation dynamics for this command
      orientationDirection : DInt := 3;   // 1: positive direction; 2: negative direction; 3: shortest distance
      bufferMode : DInt := 1;   // 1: standstill between commands, 2: blending with lower speed; 5: blending with higher speed
      transitionParameters : Array[1..5] of LReal;   // blending distance parameters
      dynamicAdaption : DInt := -1;   // <0.0: default TO setting used; 0: no dynamic adaption; 1: with variable limits; 2: with constant limits
      toolNumber : DInt;   // Tool number for SetTool command (LKINCTRL_MC_SETTOOL)
      moveDirectParameters : "LKinCtrl_typeMoveDirectParameter";   // parameters for MoveDirect command definition
      offsetParameters : "LKinCtrl_typeToolParameters";   // parameters for offset selection and configuration
      conveyorParameters : "LKinCtrl_typeConveyorParameter";   // parameters for conveyor selection and configuration
      circleParameters : "LKinCtrl_typeCircleParameters";   // parameters for circle command definition
      zoneParameters : "LKinCtrl_typeZoneParameters";   // parameters for zone commands
      pickAndPlaceParameters : "LKinCtrl_typeMovePickAndPlaceParameters";   // parameters for pick and place command
   END_STRUCT;
   // transitionParameters[1] := -1.0;
   // conveyorParameters.conveyorParaNo := 0;
END_TYPE

TYPE "LKinCtrl_typePointParameter_reduced"
   STRUCT
      pathDynamics : "LKinCtrl_typePathDynamics";   // dynamics settings for single command
      orientationDirection : DInt := 3;   // 1: positive direction; 2: negative direction; 3: shortest distance
      bufferMode : DInt := 1;   // 1: standstill between commands, 2: blending with lower speed; 5: blending with higher speed
      transitionParameters : Array[1..5] of LReal;   // blending distance parameters
      dynamicAdaption : DInt := -1;   // <0.0: default TO setting used; 0: no dynamic adaption; 1: with variable limits; 2: with constant limits
   END_STRUCT;
   // transitionParameters[1] := -1.0;
END_TYPE

TYPE "LKinCtrl_typeRelShift"
   STRUCT
      coordinates : Array[1..6] of LReal;   // Coordinates of relative CS shift
      coordinateSystem : DInt;   // Base coordinate system which shift is applied
      shiftActive : Bool;   // TRUE: Shift is active
   END_STRUCT;
END_TYPE

TYPE "LKinCtrl_typeRetProfileDist"
   STRUCT
      dist : LReal;
      functionResult : DInt;
   END_STRUCT;
END_TYPE

TYPE "LKinCtrl_typeSPTPDynamics"
   STRUCT
      velocityFactor : LReal := -1.0;   // Factor for the velocity of axis movements in relation to the respective maximum velocity of the axes. Permitted value range: -1.0 < Factor ≤ 1.0
      accelerationFactor : LReal := -1.0;   // Factor for the acceleration of axis movements in relation to the respective maximum acceleration of the axis. Permitted value range: -1.0 < Factor ≤ 1.0
      decelerationFactor : LReal := -1.0;   // Factor for the deceleration of the axis movements in relation to the respective maximum deceleration of the axis. Permitted value range: -1.0 < Factor ≤ 1.0
      jerkFactor : LReal := -1.0;   // Factor for the jerk of axis movements in relation to the respective maximum jerk of the axis. Permitted value range: -1.0 <Factor ≤ 0.0 and 0.1 < Factor ≤ 0.9
   END_STRUCT;
END_TYPE

TYPE "LKinCtrl_typeSetFlagElement_Bool"
   STRUCT
      flag : Int := -1;   // flag to be set
      flagMode : USInt := 1;   // (see LKinCtrl_PLC_Tags) 0: deactivated; 1: SET_BEFORE_AND_NO_RESET; 2: SET_BEFORE_AND_RESET_AFTER; 3: SET_BEFORE_AND_RESET_AFTER_ONE_CYCLE; 5: SET_BEFORE_AND_NO_RESET_AND_WAIT_FOR_ACKNOWLEDGE; 10: LKINCTRL_FM_SET_AT_REMAINING_DISTANCE; 11: LKINCTRL_FM_SET_AFTER_AND_NO_RESET; 13: LKINCTRL_FM_SET_AFTER_AND_RESET_AFTER_ONE_CYCLE; 15: LKINCTRL_FM_SET_AFTER_AND_NO_RESET_AND_WAIT_FOR_ACKNOWLEDGE
      remainingDistance : LReal := -1.0;   // >0.0: remainingDistance
   END_STRUCT;
END_TYPE

TYPE "LKinCtrl_typeSetFlagElement_LReal"
   STRUCT
      flag : Int := -1;   // index of flag to be set
      value : LReal := 0.0;   // value for flagValue
      flagMode : USInt := 1;   // (see LKinCtrl_PLC_Tags) 0: deactivated; 1: SET_BEFORE_AND_NO_RESET; 2: SET_BEFORE_AND_RESET_AFTER; 3: SET_BEFORE_AND_RESET_AFTER_ONE_CYCLE; 5: SET_BEFORE_AND_NO_RESET_AND_WAIT_FOR_ACKNOWLEDGE; 10: LKINCTRL_FM_SET_AT_REMAINING_DISTANCE; 11: LKINCTRL_FM_SET_AFTER_AND_NO_RESET; 13: LKINCTRL_FM_SET_AFTER_AND_RESET_AFTER_ONE_CYCLE; 15: LKINCTRL_FM_SET_AFTER_AND_NO_RESET_AND_WAIT_FOR_ACKNOWLEDGE
      remainingDistance : LReal := -1.0;   // >0.0: remainingDistance
   END_STRUCT;
END_TYPE

TYPE "LKinCtrl_typeSettings"
   STRUCT
      kinematics { ExternalAccessible := 'False'; ExternalVisible := 'False'; ExternalWritable := 'False'; S7_SetPoint := 'True'} : "LKinCtrl_typeConfigurationKinematics";
      kinematicAxes { ExternalAccessible := 'False'; ExternalVisible := 'False'; ExternalWritable := 'False'; S7_SetPoint := 'True'} : Array[1.."LKINCTRL_KINEMATICS_AXES"] of "LKinCtrl_typeConfigurationAxis";
      movePathConfiguration { ExternalAccessible := 'False'; ExternalVisible := 'False'; ExternalWritable := 'False'; S7_SetPoint := 'True'} : "LKinCtrl_typeConfiguration";
   END_STRUCT;
END_TYPE

TYPE "LKinCtrl_typeToolParameters"
   STRUCT
      offsetParaNo : Int;   // selection of offset parameter set from configuration structure
      mainPathPlane : Int;   // main path plane for compensation
   END_STRUCT;
END_TYPE

TYPE "LKinCtrl_typeWorkspaceZoneDefinition"
   STRUCT
      zoneType : DInt;   // 0:Blocked zone, 1:Work zone, 2:Signal zone
      coordinateSystem : DInt;   // 0: WCS, 1-3: OCS1-3
      frame : "LKinCtrl_typeFrame";   // shifting of the zone zero point in relation to the reference system
      geometryType : DInt;   // 0:Cuboid, 1:Sphere, 2:Cylinder
      geometryParameter : Array[1..3] of LReal;   // geometry parameter depending on geometry type
   END_STRUCT;
END_TYPE

TYPE "LKinCtrl_typeZoneParameters"
   STRUCT
      zoneConfigurationIndex : DInt;   // Index of zone configuration at MovePath
      zoneNumber : DInt;   // Zone number
      deactivationMode : DInt;   // Deactivation mode for zone commands
   END_STRUCT;
END_TYPE

TYPE "LKinCtrl_typeCOff3DPoint"
   STRUCT
      x : LReal;   // X
      y : LReal;   // Y
      z : LReal;   // Z
   END_STRUCT;
END_TYPE

TYPE "LKinCtrl_typeCOffCmdInInternal"
   STRUCT
      cmdType : Int := -1;   // 1: MoveLinAbs; 2: MoveLinRel; 3: MoveCircAbs; 4: MoveCircRel; 5: MoveDirectAbs; 6: MoveDirectRel; 10: TrackConveyorBelt; 100: WaitTime; 40/41/42: ContourOffset; 0: FlagOnlyCmd; -1: End of List
      endPoint : "LKinCtrl_typeCOff3DPoint";   // End point of command
      circleMode : DInt;   // 0: auxPoint defines point on circle line; 1: auxPoint defines circle center; 2: radius and endPoint define circle segment
      circleCenterPoint : "LKinCtrl_typeCOff3DPoint";   // Center point of circle
      circleIntermediatePoint : "LKinCtrl_typeCOff3DPoint";   // Intermediate point of circle
      circleRadius : LReal;   // Radius of circle
      circleAngle : LReal;   // Angle of circle
      pathChoice : DInt;   // circMode(0): not relevant; circMode(1): 0: pos direction; 1: neg direction; circMode(2): 0: short pos segment; 1: short neg segment; 2: long pos segment; 3: long neg segment
      circlePlane : DInt;   // circMode(0): not relevant; circMode(1+2): 0: XZ; 1: YZ; 2: XY
      transitionParameter1 : LReal;   // Transition parameter
      bufferMode : DInt;   // 1: standstill between commands, 2: blending with lower speed; 5: blending with higher speed
   END_STRUCT;
END_TYPE

TYPE "LKinCtrl_typeCOffCmdOutInternal"
   STRUCT
      cmdType : Int := -1;   // 1: MoveLinAbs; 2: MoveLinRel; 3: MoveCircAbs; 4: MoveCircRel; 5: MoveDirectAbs; 6: MoveDirectRel; 10: TrackConveyorBelt; 100: WaitTime; 40/41/42: ContourOffset; 0: FlagOnlyCmd; -1: End of List
      endPoint : "LKinCtrl_typeCOff3DPoint";   // end point of command
      circleMode : DInt;   // 0: auxPoint defines point on circle line; 1: auxPoint defines circle center; 2: radius and endPoint define circle segment
      circleCenterPoint : "LKinCtrl_typeCOff3DPoint";   // center point of circle
      circleIntermediatePoint : "LKinCtrl_typeCOff3DPoint";   // intermediate point of circle
      transitionParameter1 : LReal;   // transition parameter
      endPointOrthShifted : "LKinCtrl_typeCOff3DPoint";   // orthogonal shifted end point of command
      endPointOrthTangShifted : "LKinCtrl_typeCOff3DPoint";   // orthogonal and tangential shifted end point of command
      startPointOrthShifted : "LKinCtrl_typeCOff3DPoint";   // orthogonal shifted end point of command
      startPointOrthTangShifted : "LKinCtrl_typeCOff3DPoint";   // orthogonal and tangential shifted end point of command
      circleRadius : LReal;   // circle radius
      circleAngle : LReal;   // circle angle
      orthogonalUnitVecEnd : "LKinCtrl_typeCOff3DPoint";   // orthogonal unit vector end
      tangentialUnitVecEnd : "LKinCtrl_typeCOff3DPoint";   // tangential unit vector end
      orthogonalShiftEnd : "LKinCtrl_typeCOff3DPoint";   // orthogonal shift end
      tangentiaShiftEnd : "LKinCtrl_typeCOff3DPoint";   // tangential shift end
      orthogonalUnitVecStart : "LKinCtrl_typeCOff3DPoint";   // orthogonal unit vector start
      tangentialUnitVecStart : "LKinCtrl_typeCOff3DPoint";   // tangential unit vector start
      orthogonalShiftStart : "LKinCtrl_typeCOff3DPoint";   // orthogonal shift start
      tangentiaShiftStart : "LKinCtrl_typeCOff3DPoint";   // tangential shift start
      orthogonalUnitVecIntermediate : "LKinCtrl_typeCOff3DPoint";   // orthogonal unit vector intermediate
      tangentialUnitVecIntermediate : "LKinCtrl_typeCOff3DPoint";   // tangential unit vector intermediate
      orthogonalShiftIntermediate : "LKinCtrl_typeCOff3DPoint";   // orthogonal shift intermediate
   END_STRUCT;
END_TYPE

TYPE "LKinCtrl_typeCOffInCurrentPos"
   STRUCT
      positionAbsolute : "LKinCtrl_typeCartesianPosition";   // Source data - current absolute position
      positionAbsoluteRadComp : "LKinCtrl_typeCartesianPosition";   // Source data - current absolute position radius compensated
   END_STRUCT;
END_TYPE

TYPE "LKinCtrl_typeCOffOutNextButOneCmd"
   STRUCT
      transitionParameter : Array[1..5] of LReal;   // blending parameters
   END_STRUCT;
END_TYPE

TYPE "LKinCtrl_typeCOffPathDataOut"
   STRUCT
      nextCommand : "LKinCtrl_typePathDataElement";   // Target data - next command
      intermediateCommand : "LKinCtrl_typePathDataElement";   // Target data - intermediate (additional) command
      nextButOneCommand : "LKinCtrl_typeCOffOutNextButOneCmd";   // Target data - next but one command
      nextPositionAbsolute : "LKinCtrl_typeCartesianPosition";   // Source data - next absolute position
      nextPositionAbsoluteRadComp : "LKinCtrl_typeCartesianPosition";   // Source data - next absolute position (radius compensated)
   END_STRUCT;
   // nextCommand.cmdParameters.transitionParameters[1] := -1.0;
   // intermediateCommand.cmdParameters.transitionParameters[1] := -1.0;
END_TYPE

TYPE "LKinCtrl_typeCOffReturn"
   STRUCT
      returnValue : Word;   // Return value
      region : Int;   // Region type - see LKinCtrl_OffsetContour
      subBlockNumber : DInt;   // Sub function block number
      internalNumber : DInt;   // Internal number indicates the source code position
   END_STRUCT;
END_TYPE

TYPE "LKinCtrl_TypePnPDiagnostics"
   STRUCT
      status : Word;   // Block status
      subFunctionStatus : Word;   // Status of the subfunction
      stateNumber : DInt;   // State number
      additionalValue1 : Word;   // Additional status information
      additionalValue2 : Word;   // Additional status information
   END_STRUCT;
END_TYPE

TYPE "LKinCtrl_typePnPConveyorTracking"
   STRUCT
      enable : Bool;   // = TRUE: Set tracking with command execution
      conveyorBeltAxis : DB_ANY;   // Conveyor belt axis DB
      conveyorBeltOrigin : TO_Struct_Kinematics_Frame;   // Frame to origin of conveyor belt
      initialObjectPosition : TO_Struct_Kinematics_Frame;   // Initial object position on conveyor (only x allowed)
   END_STRUCT;
END_TYPE

TYPE "LKinCtrl_typePnPDynamics"
   STRUCT
      path : "LKinCtrl_typePathDynamics";   // Specification of the path dynamics
      orientation : "LKinCtrl_typePathDynamics";   // Specification of the orientation dynamics
      dynamicAdaption : DInt := -1;   // 0=no dynamic adaption, 1=dynamic adaptation with segmentation of the path, 2=dynamic adaptation without segmentation of the path
   END_STRUCT;
END_TYPE

TYPE "LKinCtrl_typePnPInitTOData"
   STRUCT
      factorBlendingLength : LReal;   // Factor blending length
      orientationDefaults : "LKinCtrl_typePathDynamics";   // Orientation default dynamics
   END_STRUCT;
END_TYPE

TYPE "LKinCtrl_typePnPLinCmdSeqParameter"
   STRUCT
      start : "LKinCtrl_typePnPLinPointParameter";   // Parameter for start position
      postStart : "LKinCtrl_typePnPLinPointParameter";   // Parameter for post start motion
      intermediate : "LKinCtrl_typePnPLinPointParameter";   // Parameter for intermediate motion
      preTarget : "LKinCtrl_typePnPLinPointParameter";   // Parameter for pre target motion
      target : "LKinCtrl_typePnPLinPointParameter";   // Parameter for target motion
      numberOfUsedCmd : DInt;   // Number of used commands
   END_STRUCT;
   // start.transitionParameter[1] := -1.0;
   // postStart.transitionParameter[1] := -1.0;
   // intermediate.transitionParameter[1] := -1.0;
   // preTarget.transitionParameter[1] := -1.0;
   // target.transitionParameter[1] := -1.0;
END_TYPE

TYPE "LKinCtrl_typePnPLinPointParameter"
   STRUCT
      usePoint : Bool;   // Use or ignore point
      position : Array[1..6] of LReal;   // Cartesian position
      coordSystem : DInt;   // 0: WCS; 1: OCS[1]; 2: OCS[2]; 3: OCS[3]; 100: MCS
      bufferMode : DInt := 1;   // bufferMode for path motion
      transitionParameter : Array[1..5] of LReal;   // transitionParameter for path motion
      tracking : "LKinCtrl_typePnPTrackingProperties";   // Tracking properties
      directionA : DInt := 3;   // 1 - positive, 2 - negative, 3 - shortest way (Only necessary up to 4D Kinematics)
      pathDynamics : "LKinCtrl_typePathDynamics";   // Path dynamics specification
      dynamicAdaption : DInt;   // 0=no dynamic adaption, 1=dynamic adaptation with segmentation of the path, 2=dynamic adaptation without segmentation of the path
      distanceToPrevious : LReal;   // Linear distance to previous point
   END_STRUCT;
   // transitionParameter[1] := -1.0;
END_TYPE

TYPE "LKinCtrl_typePnPOrientationFrame"
   STRUCT
      "a" : LReal;   // Orientation A
      "b" : LReal;   // Orientation B
      c : LReal;   // Orientation C
   END_STRUCT;
END_TYPE

TYPE "LKinCtrl_typePnPParameter"
   STRUCT
      direction : Array[1..3] of LReal;   // Direction of vector (will be normed by FB) from start / target
      workingHeight : LReal := 0.0;   // Length of vector
      transitionArea : LReal := 0.0;   // Permissible blending area at end of vector
      dynamicsFactor : LReal := 100.0;   // Path dynamics scaling factor
   END_STRUCT;
END_TYPE

TYPE "LKinCtrl_typePnPTrackingProperties"
   STRUCT
      active : Bool;   // TRUE: Tracking is active
      velocity : LReal;   // Velocity of OCS
      frame : "LKinCtrl_typeFrame";   // Base frame of OCS
      objectPosition : "LKinCtrl_typeFrame";   // Relative OCS shift in base frame
   END_STRUCT;
END_TYPE

DATA_BLOCK "GDB_HMI_Status"   // DB13
TITLE = HMI status facade DB (read-only, Phase 2.4)
{ S7_Optimized_Access := 'TRUE' }
// Phase 2.4 (C71, 2026-05-18) — Read-only HMI facade. Consolidates ~35 display tags from across the system (GDB_Control, GDB_ManualStatus, GDB_MachineCmd, GDB_PalletizingCmd, instFB_AutoCtrl_ABCDE iDB, instFB_AutoCtrl_Palletizing iDB, J{n}_SCARA_Arm3D TOs, instFB_AxisCtrl iDB) into a single GDB for HMI to bind to. FB_HMIStatusMirror updates this each OB1 scan via active-mode routing logic. Writes (HMI → bo_Mode/bo_Start/etc.) stay direct to the per-mode cmd DBs — this GDB is read-only from HMI's perspective.
// stored: MemoryReserve 100
   VAR
      activeMode : Int;   // Active cycle mode: 0=None, 1=ABCDE, 2=Palletizing, 3=Manual. Derived each scan from the 3 GDB_*Cmd.bo_Mode bits (set by HMI/operator). PLC mutex contract: only one mode may have Start succeed at a time. HMI may bind this to a banner text/lamp.
      currentStep : Int;   // Mode-routed current step. activeMode=1: mirrors GDB_MachineCmd.i16_AutoStep (0,10..50). activeMode=2: mirrors GDB_PalletizingCmd.i16_PalletStep (0..48). activeMode=3: 0 (manual has no step). activeMode=0: 0.
      totalSteps : Int;   // Total steps in active cycle: 5 (ABCDE), 48 (Palletizing), 0 (Manual/None). HMI uses for progress-bar / "Step N of M" display.
      target_x : LReal;   // Current TCP target X (mm), mode-routed. ABCDE: instFB_AutoCtrl_ABCDE.statTargetPos.x. Palletizing: instFB_AutoCtrl_Palletizing.statTargetPos.x. Manual/None: holds last value (no overwrite, so HMI sees last commanded target).
      target_y : LReal;   // Current TCP target Y (mm), mode-routed. See target_x.
      target_z : LReal;   // Current TCP target Z (mm), mode-routed. See target_x.
      target_a : LReal;   // Current TCP target A wrist (deg), mode-routed. See target_x.
      axesEnabled : Bool;   // Group: all 4 joints powered. Mirror of GDB_Control.axesEnabled.
      axesHomed : Bool;   // Group: all 4 joints homed. Mirror of GDB_Control.axesHomed.
      axesError : Bool;   // Group: any joint error. Mirror of GDB_Control.axesError.
      axesReady : Bool;   // Group: enabled AND homed AND NOT error. Mirror of GDB_Control.axesReady (derived in FB_AxisCtrl rev 1.3).
      j1_enabled : Bool;   // J1 base shoulder: ready / powered. Mirror of GDB_ManualStatus.bo_J1_Enabled (which mirrors instFB_AxisCtrl.instPower_J1.Status).
      j1_homed : Bool;   // J1: homed (mirror of J1_SCARA_Arm3D.StatusWord.%X5 via GDB_ManualStatus).
      j1_error : Bool;   // J1: fault active.
      j1_jogActive : Bool;   // J1: motion in progress (NOT standstill).
      j1_actualPos : LReal;   // J1 actual position (degrees, base shoulder rotation). Read direct from J1_SCARA_Arm3D.ActualPosition.
      j1_actualVel : LReal;   // J1 actual velocity (deg/s).
      j2_enabled : Bool;
      j2_homed : Bool;
      j2_error : Bool;
      j2_jogActive : Bool;
      j2_actualPos : LReal;   // J2 elbow actual rotation (degrees). NOTE: J2 is at kinematic-group index A[3] per the deliberate misorder — see PLC_HANDOFF_2026-05-18_J2J3DeliberateMisorder.md. This field reads from J2_SCARA_Arm3D.ActualPosition directly (joint-name convention, no swap needed here).
      j2_actualVel : LReal;
      j3_enabled : Bool;
      j3_homed : Bool;
      j3_error : Bool;
      j3_jogActive : Bool;
      j3_actualPos : LReal;   // J3 Z prismatic actual position (mm). NOTE: J3 is at kinematic-group index A[2] per the deliberate misorder. This field reads from J3_SCARA_Arm3D.ActualPosition (joint-name convention).
      j3_actualVel : LReal;
      j4_enabled : Bool;
      j4_homed : Bool;
      j4_error : Bool;
      j4_jogActive : Bool;
      j4_actualPos : LReal;   // J4 wrist actual rotation (degrees).
      j4_actualVel : LReal;
      estopLock : Bool;   // Safety: E-Stop chain healthy (mirror of GDB_MachineCmd.bo_ESTOP_LOCK). TRUE=OK, FALSE=E-Stop active.
      alarm : Bool;   // Aggregate alarm: GDB_MachineCmd.bo_Alarm OR GDB_PalletizingCmd.bo_Alarm. HMI binds a single lamp to this for "any alarm" indication.
      pathInitialed : Bool;   // ABCDE 5-point path is initialized (mirror of GDB_MachineCmd.bo_PathInitialed). Required gate before ABCDE Start.
      palletInitialed : Bool;   // Palletizing 16-box 4-layer path is initialized (mirror of GDB_PalletizingCmd.bo_PalletInitialed). Required gate before Palletizing Start.
      toolActive : Bool;   // Diagnostic: MC_SetTool(ToolNumber=1) has been activated on ScaraArm3D (mirror of instFB_AxisCtrl.statToolActivated). FALSE → MC_MoveLinearAbsolute returns UserFault (motionFBStatus=0x8001). FB_AxisCtrl rev 1.2+ auto-fires SetTool once after axesEnabled goes TRUE.
   END_VAR
BEGIN
END_DATA_BLOCK

DATA_BLOCK "GDB_MCDData"   // DB6
{ S7_Optimized_Access := 'TRUE' }
// stored: MemoryReserve 100
   VAR
      Velocity : Array[1..4] of LReal;   // Kinematic-group view of per-axis velocity (from ScaraArm3D.AxesData.A[i].Velocity). Used by NX MCD via signal adapters.
      Position : Array[1..4] of LReal;   // Kinematic-group view of per-axis position (from ScaraArm3D.AxesData.A[i].Position). Used by NX MCD via signal adapters.
      J1_ActualPosition : LReal;   // Phase C.0 (2026-05-17): direct mirror of J1_SCARA_Arm3D.ActualPosition (TO_Axis attribute). Exists for PLCSIM-Adv API monitoring (TO_Axis tags not exposed via API directly; HMI runtime uses TIA S7 driver which can read them). DIAGNOSTIC MIRROR — HMI continues to bind to J1_SCARA_Arm3D.ActualPosition direct.
      J1_ActualVelocity : LReal;   // Phase C.0 (2026-05-17): direct mirror of J1_SCARA_Arm3D.ActualVelocity. See J1_ActualPosition comment.
      J2_ActualPosition : LReal;   // Phase C.0 (2026-05-17): direct mirror of J2_SCARA_Arm3D.ActualPosition. See J1_ActualPosition comment.
      J2_ActualVelocity : LReal;   // Phase C.0 (2026-05-17): direct mirror of J2_SCARA_Arm3D.ActualVelocity. See J1_ActualPosition comment.
      J3_ActualPosition : LReal;   // Phase C.0 (2026-05-17): direct mirror of J3_SCARA_Arm3D.ActualPosition. See J1_ActualPosition comment.
      J3_ActualVelocity : LReal;   // Phase C.0 (2026-05-17): direct mirror of J3_SCARA_Arm3D.ActualVelocity. See J1_ActualPosition comment.
      J4_ActualPosition : LReal;   // Phase C.0 (2026-05-17): direct mirror of J4_SCARA_Arm3D.ActualPosition. See J1_ActualPosition comment.
      J4_ActualVelocity : LReal;   // Phase C.0 (2026-05-17): direct mirror of J4_SCARA_Arm3D.ActualVelocity. See J1_ActualPosition comment.
      BeltVelocity : LReal;   // Phase D.0 (2026-05-19): conveyor belt velocity command to MCD (PLC writes, MCD reads via sContainerBeltVel signal adapter on saContainerBe... owner). Unit: mm/s. Set by FB_ConveyorCtrl (future) or operator Watch Table for now. Default 0.0 (belt stopped).
      SpawnContainerCmd : Bool;   // Phase D.0 (2026-05-19): trigger to spawn a new container in MCD physics scene (PLC writes rising-edge pulse, MCD reads via sActivateSpawnContainer signal adapter on saContainerBe... owner). Each rising edge spawns one container at the source position. Used by FB_Palletizing test harness or operator override.
      SinkContainerLeft : Bool;   // Phase D.0 (2026-05-19): trigger to remove container at LEFT sink position (PLC writes rising-edge pulse, MCD reads via sSinkContainer signal on saContainerPallet_1 OR _2 — operator picks which physical adapter corresponds to "left" at TIA mapping step). Rising edge removes one container. V3.0 cycle does not actively drive sinks; reserve for V3.1+ pallet-full cleanup logic.
      SinkContainerRight : Bool;   // Phase D.0 (2026-05-19): trigger to remove container at RIGHT sink position (PLC writes rising-edge pulse, MCD reads via sSinkContainer signal on the other saContainerPallet_X). Operator's pairing decision at TIA mapping step. V3.0 cycle does not actively drive sinks; reserve for V3.1+.
      PackingSensor : Bool;   // Phase D.0 (2026-05-19): container-reached-packing-position sensor (MCD writes via sContainerBeltPackingSensor signal adapter on saContainerBe... owner, PLC reads). TRUE when a container is detected at the packing station; used by FB_ConveyorCtrl (future) to advance the state machine to "container ready for ABCDE pick" or operator visual confirmation.
      PalletizingSensor : Bool;   // Phase D.0 (2026-05-19): container-reached-palletizing-position sensor (MCD writes via sContainerBeltPalletizingSensor signal adapter on saContainerBe... owner, PLC reads). TRUE when a container is detected at the palletizing station; used by FB_AutoCtrl_Palletizing (future) to gate the pick-and-place cycle on actual container arrival vs free-running cycle.
      BeltStopperSensor : Bool;   // Phase D.2 (2026-05-19): belt mechanical stopper active state (MCD writes via sContainerBeltStopperSensor signal adapter on saContainerBelt_1 owner, PLC reads). TRUE = stopper is engaged (mechanically blocking belt flow); FALSE = released. Provides redundant arrival confirmation alongside PalletizingSensor, and diagnostic feedback if stopper sticks in either state. V3.0 cycle doesn't strictly require this (uses PalletizingSensor as pick gate), but operator can monitor it via Watch Table during smoke runs.
      SpawnContainerCompleteCmd : Bool;   // Phase D.1 (2026-05-19): trigger to spawn a pre-completed/stacked container variant in MCD (PLC writes rising-edge pulse, MCD reads). Maps to NX Object Source `objsrcContainerComplete_1`. Unused in V3.0 base orchestration; reserve for V3.1+ recipe-driven box variants (e.g., different sizes, pre-stacked pallet demo).
      SinkContainerBelt : Bool;   // Phase D.1 (2026-05-19): trigger to remove container at conveyor end-of-line / generic sink position (PLC writes, MCD reads). Maps to NX Object Sink `objsinkContainer_1`. Distinct from SinkContainerLeft/Right which are pallet-specific. Unused in V3.0; reserve for V3.1+ conveyor cleanup (e.g., reject lane, end-of-line discard).
      SinkContainerSensor : Bool;   // Phase D.1 (2026-05-19): sink-zone collision sensor (MCD writes via csContainerSink_1 collision-sensor signal, PLC reads). TRUE when a container is detected entering the sink zone. Reserve for V3.1+ confirm-removal feedback (FB verifies SCARA actually dropped the box rather than just commanding release).
      ScaraHasGrippedObj : Bool;   // Grip-success feedback (2026-05-21): MCD writes via the sScaraHasGrippedObj output signal on the Suction_Cup_Gripper SignalAdapter (MCD writes, PLC reads). TRUE = the suction cup has successfully gripped a container; FALSE = nothing held. Lets the PLC confirm a real pick before the SCARA raises, and pins the grip chain for diagnostics.
   END_VAR
BEGIN
END_DATA_BLOCK

DATA_BLOCK "GDB_Control"   // DB
TITLE = GDB_Control (minimal)
{ S7_Optimized_Access := 'TRUE' }
// Minimal control DB for ABCDE 5-point cycle. Holds kinematic enable/home arrays + mirror status. Trimmed from v9 (palletizing/recipe/manual fields removed).
   VAR
      enableAxes : Bool;   // Enable kinematic group via LKinCtrl_MC_GroupPower
      axesEnabled : Bool;   // Status: all axes enabled (mirror from MC_GroupPower.axesEnabled)
      resetAxes : Bool;   // Reset kinematic group via LKinCtrl_MC_GroupReset
   END_VAR
   VAR RETAIN
      axesError : Bool;   // Status: error on any joint TO
   END_VAR
   VAR
      homeAxes : Bool;   // Home kinematic group via LKinCtrl_MC_GroupHome
      axesHomed : Bool;   // Status: all 4 joint TOs report StatusWord.X5 (Homed)
      robotStandstill : Bool;   // Status: all 4 joint TOs report StatusWord.X7 (Standstill)
   END_VAR
   VAR RETAIN
      HomePos : Array[1..6] of LReal;   // Home positions per kinematic axis index (A1=J1, A2=J3, A3=J2, A4=J4). Initialized by Startup.scl.
   END_VAR
   VAR
      HomeMode : Array[1..6] of Int;   // Home mode per kinematic axis index. 7 = set actual position (no physical homing motion).
      StartMode : Array[1..6] of DInt;   // Start mode for MC_Power per axis. 1 = enable position-controlled. Initialized by Startup.scl to avoid retain-drift issues.
      StopMode : Array[1..6] of Int;   // Stop mode for MC_Power per axis. 1 = immediate stop. Initialized by Startup.scl.
      RestartMode : Array[1..7] of Bool;   // Restart mode flags for MC_GroupReset per axis.
   END_VAR
BEGIN
END_DATA_BLOCK

DATA_BLOCK "GDB_MachineCmd"   // DB
TITLE = Machine command/status DB
{ S7_Optimized_Access := 'TRUE' }
// Wang Shuo / Huashili-style command + status struct for ABCDE auto cycle. HMI binds buttons here.
   VAR
      bo_InitPath : Bool;   // HMI: rising edge → initialize ABCDE 5-point path data / HMI: 上升沿 → 初始化 ABCDE 5 点路径
      bo_Start : Bool;   // HMI: rising edge → start auto cycle (i16_AutoStep := 10) / HMI: 上升沿 → 启动自动循环
      bo_Stop : Bool;   // HMI: rising edge → stop auto cycle (i16_AutoStep := 0) / HMI: 上升沿 → 停止自动循环
      bo_Mode : Bool := TRUE;   // HMI: AUTO mode selector (TRUE = auto cycle enabled, FALSE = ignored) / HMI: 自动模式开关
      bo_ESTOP_LOCK : Bool := TRUE;   // Safety: E-Stop chain healthy (TRUE = OK, FALSE = E-Stop active) / 安全: 急停健康状态
      bo_PathInitialed : Bool;   // Status: ABCDE path has been initialized (set after bo_InitPath rising edge) / 状态: 路径已初始化
      bo_Alarm : Bool;   // Status: any system alarm (placeholder, always FALSE in minimal demo) / 状态: 系统报警
      i16_AutoStep : Int;   // Main state machine step. 6-state per source spec 杨子楠5月17日周计划.md §3.3: 0=idle, 10=going-to-A, 20=going-to-B, 30=going-to-C, 40=going-to-D, 50=going-to-E. Cycle wraps 50→10 (source spec §3.5). Wang Shuo / Huashili 4-REGION pattern. / 主状态机步号 (6 状态, 来源 §3.3): 0=空闲, 10=去A, 20=去B, 30=去C, 40=去D, 50=去E. 循环 50→10 (§3.5). 王硕模式
   END_VAR
BEGIN
END_DATA_BLOCK

DATA_BLOCK "GDB_ManualCmd"   // DB
TITLE = Manual-mode command DB (Phase G)
{ S7_Optimized_Access := 'TRUE' }
// Phase G (C67, 2026-05-18) — Manual-mode command surface. Sibling to GDB_MachineCmd (auto) + GDB_Control (axis-group). HMI binds the 20 per-axis cmd buttons + 4 Kin target IOFields + 4 Kin group buttons here. FB_ManualCtrl on OB30 (10ms cyclic) consumes these and routes to MC_MoveJog / MC_MoveLinearAbsolute / GDB_Control flags.
   VAR
      bo_Mode : Bool := FALSE;   // HMI: Manual mode selector (TRUE = manual cmds active, FALSE = ignored). Mutex with GDB_MachineCmd.bo_Mode — operator must turn AUTO off before enabling MANUAL. FB_ManualCtrl REGION 1 gates all manual actions on (bo_Mode AND bo_ESTOP_LOCK AND NOT GDB_MachineCmd.bo_Mode). / HMI: 手动模式开关 (与 AUTO 模式互斥)
      bo_ESTOP_LOCK : Bool := TRUE;   // Safety: E-Stop chain healthy (TRUE = OK, FALSE = E-Stop active). Mirrors GDB_MachineCmd.bo_ESTOP_LOCK convention. / 安全: 急停健康状态
      bo_J1_Enable : Bool;   // HMI manual: J1 Enable button. Routes via FB_ManualCtrl REGION 2 to GDB_Control.enableAxes (group-level; enabling J1 enables all 4 joints together — see PLC_HANDOFF_2026-05-18_C67 §Risk-7). / HMI 手动: J1 使能 (实际为整组使能)
      bo_J2_Enable : Bool;   // HMI manual: J2 Enable button (routes to group). See bo_J1_Enable.
      bo_J3_Enable : Bool;   // HMI manual: J3 Enable button (routes to group). See bo_J1_Enable.
      bo_J4_Enable : Bool;   // HMI manual: J4 Enable button (routes to group). See bo_J1_Enable.
      bo_J1_Home : Bool;   // HMI manual: J1 Home button. Routes via FB_ManualCtrl REGION 2 to GDB_Control.homeAxes (group-level; sets all 4 joint actuals to HomePos via MC_Home Mode=7). / HMI 手动: J1 回零 (实际为整组回零)
      bo_J2_Home : Bool;   // HMI manual: J2 Home button (routes to group).
      bo_J3_Home : Bool;   // HMI manual: J3 Home button (routes to group).
      bo_J4_Home : Bool;   // HMI manual: J4 Home button (routes to group).
      bo_J1_Reset : Bool;   // HMI manual: J1 Reset button. Routes via FB_ManualCtrl REGION 2 to GDB_Control.resetAxes (group-level; pulses MC_Reset on all 4 joints + kin TO). / HMI 手动: J1 复位 (实际为整组复位)
      bo_J2_Reset : Bool;   // HMI manual: J2 Reset button (routes to group).
      bo_J3_Reset : Bool;   // HMI manual: J3 Reset button (routes to group).
      bo_J4_Reset : Bool;   // HMI manual: J4 Reset button (routes to group).
      bo_J1_JogForward : Bool;   // HMI manual: J1 Jog-Forward HOLD button (level-triggered). FB_ManualCtrl REGION 3 routes via XOR safety to MC_MoveJog.JogForward on J1_SCARA_Arm3D at 10°/s default. Releasing the button decelerates to standstill. / HMI 手动: J1 正向点动 (按住)
      bo_J1_JogBackward : Bool;   // HMI manual: J1 Jog-Backward HOLD button (level-triggered). See bo_J1_JogForward. If both forward + backward held simultaneously, XOR safety in REGION 3 makes neither direction win. / HMI 手动: J1 反向点动 (按住)
      bo_J2_JogForward : Bool;   // HMI manual: J2 Jog-Forward HOLD button. See bo_J1_JogForward.
      bo_J2_JogBackward : Bool;   // HMI manual: J2 Jog-Backward HOLD button. See bo_J1_JogBackward.
      bo_J3_JogForward : Bool;   // HMI manual: J3 Jog-Forward HOLD button. See bo_J1_JogForward.
      bo_J3_JogBackward : Bool;   // HMI manual: J3 Jog-Backward HOLD button. See bo_J1_JogBackward.
      bo_J4_JogForward : Bool;   // HMI manual: J4 Jog-Forward HOLD button. See bo_J1_JogForward.
      bo_J4_JogBackward : Bool;   // HMI manual: J4 Jog-Backward HOLD button. See bo_J1_JogBackward.
      cfgKinTargetX : LReal := 1500.0;   // HMI manual: operator-set Kin target X coordinate (mm in WCS). Consumed by FB_ManualCtrl REGION 4 on bo_KinGo rising edge, passed to MC_MoveLinearAbsolute on ScaraArm3D. StartValue 1500.0 = ABCDE A-point safe default. / HMI 手动: 运动学目标 X 坐标 (mm)
      cfgKinTargetY : LReal := 300.0;   // HMI manual: operator-set Kin target Y coordinate (mm in WCS). See cfgKinTargetX. / HMI 手动: 运动学目标 Y 坐标 (mm)
      cfgKinTargetZ : LReal := 400.0;   // HMI manual: operator-set Kin target Z coordinate (mm in WCS). See cfgKinTargetX. / HMI 手动: 运动学目标 Z 坐标 (mm)
      cfgKinTargetA : LReal := 0.0;   // HMI manual: operator-set Kin target A orientation (degrees). See cfgKinTargetX. / HMI 手动: 运动学目标 A 姿态 (度)
      bo_KinGo : Bool;   // HMI manual: rising-edge → trigger MC_MoveLinearAbsolute on ScaraArm3D to (cfgKinTargetX, Y, Z, A). FB_ManualCtrl REGION 4 uses BufferMode=0 (aborting) for clean handoff from any in-flight auto motion. / HMI 手动: 上升沿 → 执行运动学绝对移动
      bo_KinEnable : Bool;   // HMI manual: Kin-group Enable button. Routes via FB_ManualCtrl REGION 2 to GDB_Control.enableAxes. Functionally equivalent to bo_J1_Enable (group-level wiring). / HMI 手动: 运动学组使能
      bo_KinHome : Bool;   // HMI manual: Kin-group Home button. Routes via FB_ManualCtrl REGION 2 to GDB_Control.homeAxes. / HMI 手动: 运动学组回零
      bo_KinReset : Bool;   // HMI manual: Kin-group Reset button. Routes via FB_ManualCtrl REGION 2 to GDB_Control.resetAxes. / HMI 手动: 运动学组复位
   END_VAR
BEGIN
END_DATA_BLOCK

DATA_BLOCK "GDB_ManualStatus"   // DB
TITLE = Manual-mode status DB (Phase G)
{ S7_Optimized_Access := 'TRUE' }
// Phase G (C67, 2026-05-18) — Manual-mode status mirror (PLC sole writer; HMI binds for BackColor lamps + R/O text fields). Per HMI cycle-7.1 BackColor Q&A Option A: clean PLC-side mirror (typed Bool members) preferred over runtime bit-mask of TO_Axis StatusWord (WinCC Unified Basic PlcTag does not support %X{n} bit-slice paths).
   VAR
      bo_J1_Enabled : Bool;   // PLC-derived: J1 axis is enabled / ready (mirror of J1_SCARA_Arm3D.StatusWord.%X3 — production-canonical Ready bit per v9 FB_AxisManualWiring). Set by FB_ManualCtrl REGION 5 (status mirror). / PLC 衍生: J1 使能/就绪状态
      bo_J2_Enabled : Bool;   // PLC-derived: J2 axis is enabled / ready (mirror of J2_SCARA_Arm3D.StatusWord.%X3).
      bo_J3_Enabled : Bool;   // PLC-derived: J3 axis is enabled / ready (mirror of J3_SCARA_Arm3D.StatusWord.%X3).
      bo_J4_Enabled : Bool;   // PLC-derived: J4 axis is enabled / ready (mirror of J4_SCARA_Arm3D.StatusWord.%X3).
      bo_J1_Homed : Bool;   // PLC-derived: J1 axis is homed (mirror of J1_SCARA_Arm3D.StatusWord.%X5 — per ABCDE GDB_Control.axesHomed convention). / PLC 衍生: J1 已回零
      bo_J2_Homed : Bool;   // PLC-derived: J2 axis is homed (mirror of J2_SCARA_Arm3D.StatusWord.%X5).
      bo_J3_Homed : Bool;   // PLC-derived: J3 axis is homed (mirror of J3_SCARA_Arm3D.StatusWord.%X5).
      bo_J4_Homed : Bool;   // PLC-derived: J4 axis is homed (mirror of J4_SCARA_Arm3D.StatusWord.%X5).
      bo_J1_Error : Bool;   // PLC-derived: J1 axis has fault (mirror of J1_SCARA_Arm3D.StatusWord.%X1 — per v9 axesError convention). / PLC 衍生: J1 故障
      bo_J2_Error : Bool;   // PLC-derived: J2 axis has fault (mirror of J2_SCARA_Arm3D.StatusWord.%X1).
      bo_J3_Error : Bool;   // PLC-derived: J3 axis has fault (mirror of J3_SCARA_Arm3D.StatusWord.%X1).
      bo_J4_Error : Bool;   // PLC-derived: J4 axis has fault (mirror of J4_SCARA_Arm3D.StatusWord.%X1).
      bo_J1_JogActive : Bool;   // PLC-derived: J1 axis is moving (NOT StatusWord.%X7 standstill — derived as "non-standstill"). Useful for HMI to lit a "moving" lamp during jog. / PLC 衍生: J1 在运动中
      bo_J2_JogActive : Bool;   // PLC-derived: J2 axis is moving (NOT StatusWord.%X7).
      bo_J3_JogActive : Bool;   // PLC-derived: J3 axis is moving (NOT StatusWord.%X7).
      bo_J4_JogActive : Bool;   // PLC-derived: J4 axis is moving (NOT StatusWord.%X7).
      bo_KinEnabled : Bool;   // PLC-derived: kinematic group is enabled (mirror of GDB_Control.axesEnabled — aggregated 4-joint Power.Status from FB_AxisCtrl REGION Power). / PLC 衍生: 运动学组使能
      bo_KinReady : Bool;   // PLC-derived: kinematic group is ready (mirror of GDB_Control.axesReady = axesEnabled AND axesHomed AND NOT axesError). Per HMI cycle-7.1 BackColor Q&A — single Bool tag enables Range-dyn lamp binding without bit-mask workaround. / PLC 衍生: 运动学组就绪
      bo_KinHomed : Bool;   // PLC-derived: kinematic group is homed (mirror of ScaraArm3D.StatusWord.%X5). / PLC 衍生: 运动学组已回零
      bo_KinError : Bool;   // PLC-derived: kinematic group has fault (ScaraArm3D.ErrorWord <> 0). Aggregates all per-axis + kinematic-specific errors. / PLC 衍生: 运动学组故障
      bo_KinManualBusy : Bool;   // PLC-derived: manual Kin MC_MoveLinearAbsolute is in flight (mirror of instMoveLinAbs.Busy in FB_ManualCtrl REGION 4). HMI uses for "Manual move busy" lamp during point-to-point motion. / PLC 衍生: 手动绝对移动忙
   END_VAR
BEGIN
END_DATA_BLOCK

DATA_BLOCK "GDB_PalletizingCmd"   // DB
TITLE = Palletizing command/status DB (C69 Phase 2.2)
{ S7_Optimized_Access := 'TRUE' }
// Wang Shuo / Huashili-style command + status struct for C69 Phase 2.2 16-box 4-layer palletizing cycle. Sibling DB to GDB_MachineCmd (ABCDE 5-point) and GDB_ManualCmd (manual mode, STAGED_FOR_PHASE_2). HMI binds palletizing buttons here. Mode arbitration via 3-way mutex: GDB_MachineCmd.bo_Mode XOR GDB_PalletizingCmd.bo_Mode XOR GDB_ManualCmd.bo_Mode.
   VAR
      bo_InitPallet : Bool;   // HMI: rising edge -> initialize 16-box 4-layer palletizing path (path runs from box 1 layer 1 through box 16 layer 4, 3 phases per box approach/place/retract) / HMI: 上升沿 -> 初始化 16 箱 4 层码垛路径
      bo_Start : Bool;   // HMI: rising edge -> start palletizing cycle (i16_PalletStep := 1). Permissive checks: bo_Mode AND bo_ESTOP_LOCK AND bo_PalletInitialed AND NOT bo_Alarm AND NOT GDB_MachineCmd.bo_Mode (ABCDE mutex) AND NOT GDB_ManualCmd.bo_Mode (manual mutex). / HMI: 上升沿 -> 启动码垛循环
      bo_Stop : Bool;   // HMI: rising edge -> stop palletizing cycle (i16_PalletStep := 0) / HMI: 上升沿 -> 停止码垛循环
      bo_Mode : Bool := FALSE;   // HMI: Palletizing AUTO mode selector (TRUE = palletizing cycle enabled, FALSE = ignored). Mutually exclusive with GDB_MachineCmd.bo_Mode (ABCDE cycle) and GDB_ManualCmd.bo_Mode (manual). Operator must turn other modes off before enabling palletizing. / HMI: 码垛自动模式开关 (与 ABCDE 和 手动模式互斥)
      bo_ESTOP_LOCK : Bool := TRUE;   // Safety: E-Stop chain healthy (TRUE = OK, FALSE = E-Stop active). Mirrors GDB_MachineCmd.bo_ESTOP_LOCK convention. / 安全: 急停健康状态
      bo_PalletInitialed : Bool;   // Status: 16-box 4-layer palletizing path has been initialized (set after bo_InitPallet rising edge inside FB_AutoCtrl_Palletizing REGION 1) / 状态: 码垛路径已初始化
      bo_Alarm : Bool;   // Status: any palletizing-specific alarm (placeholder; always FALSE in C69 Phase 2.2 demo) / 状态: 码垛报警
      i16_PalletStep : Int;   // Main palletizing state machine. 0 = idle, 1..48 = active path point (16 boxes x 3 phases). Step encoding: box_index = ((step-1) DIV 3) + 1; phase = ((step-1) MOD 3) + 1 [1=approach, 2=place, 3=retract]. Cycle wraps 48 -> 1. Layer = ((box_index-1) DIV 4) + 1 (4 layers, 4 boxes per layer). / 码垛主状态: 0=空闲, 1..48=路径点 (16箱 x 3阶段 = 4层 x 4箱/层 x 3阶段). 循环 48->1
      i16_TotalBoxes : Int := 16;   // C69 Phase 2.2 (2026-05-18): hardcoded 16-box pattern = 4 layers x 4 boxes/layer x 3 phases = 48 path points. Mirrors statActiveBoxes from FB_AutoCtrl_Palletizing iDB (snapshotted at last InitPallet pulse). V3.x recipe-driven would change this; for V2 hardcoded port, always 16. / 总箱数 (V2 硬编码 16): 4 层 x 4 箱/层 x 3 阶段 = 48 路径点
   END_VAR
BEGIN
END_DATA_BLOCK

DATA_BLOCK "GDB_PalletizingPath"   // DB
TITLE = Palletizing buffered-path command list (V4.0)
{ S7_Optimized_Access := 'TRUE' }
// Buffered-path command list for the V4.0 palletizing executor. Array of UDT_PathCmd, built once per bo_InitPallet rising edge and executed by FB_AutoCtrl_Palletizing REGION 4. Kept as a separate global DB (not an instance-DB stat array) so the PowerShell smoke harness can probe aCmd[n] directly.
   VAR
      aCmd : Array[1..200] of "UDT_PathCmd";   // Buffered-path command list -- built by FB_AutoCtrl_Palletizing REGION 1 (9 commands per box x 16 boxes + 1 END_OF_PATH ~= 145 used) and walked by the REGION 4 executor. [1..200] gives headroom.
      i16_CmdCount : Int;   // Number of valid commands in aCmd, set by REGION 1 after building the list. The END_OF_PATH command sits at aCmd[i16_CmdCount].
   END_VAR
BEGIN
END_DATA_BLOCK

DATA_BLOCK "GDB_AxisCtrl"   // DB101
{ S7_Optimized_Access := 'TRUE' }
// stored: AutoNumber false, MemoryReserve 0
   VAR
      TOCtrl { S7_SetPoint := 'True'} : Array[1..10] of "UDT_typePosCtrl";
      LKinCtrl { S7_SetPoint := 'True'} : "UDT_typeKinCtrl";
      Measureinput { S7_SetPoint := 'True'} : Array[1..2] of "UDT_typeMeasureInput";
   END_VAR
BEGIN
   LKinCtrl.input.configuration.jogframe.dynamics.path.velocity := 200.0;
   LKinCtrl.input.configuration.jogframe.dynamics.path.acceleration := 2000.0;
   LKinCtrl.input.configuration.jogframe.dynamics.path.deceleration := 2000.0;
   LKinCtrl.input.configuration.jogframe.dynamics.path.jerk := 20000.0;
   LKinCtrl.input.configuration.jogframe.dynamics.orientation.velocity := 50.0;
   LKinCtrl.input.configuration.jogframe.dynamics.orientation.acceleration := 500.0;
   LKinCtrl.input.configuration.jogframe.dynamics.orientation.deceleration := 500.0;
   LKinCtrl.input.configuration.jogframe.dynamics.orientation.jerk := 5000.0;
END_DATA_BLOCK

